LIN {X 0,Y 530.972,Z 518.34,A -85,B 0,C 180,E1 -4177.507,E2 -4177.507} C_VEL
LIN {X 0,Y 530.988,Z 518.342,A -85,B 0,C 180,E1 -4180.433,E2 -4180.433} C_VEL
LIN {X 0,Y 530.965,Z 518.332,A -85,B 0,C 180,E1 -4183.281,E2 -4183.281} C_VEL
LIN {X 0,Y 530.993,Z 518.336,A -85,B 0,C 180,E1 -4185.621,E2 -4185.621} C_VEL
LIN {X 0,Y 531.003,Z 518.341,A -85,B 0,C 180,E1 -4188.565,E2 -4188.565} C_VEL
LIN {X 0,Y 530.963,Z 518.337,A -85,B 0,C 180,E1 -4191.529,E2 -4191.529} C_VEL
LIN {X 0,Y 530.959,Z 518.348,A -85,B 0,C 180,E1 -4194.38,E2 -4194.38} C_VEL
LIN {X 0,Y 530.972,Z 518.342,A -85,B 0,C 180,E1 -4197.133,E2 -4197.133} C_VEL
LIN {X 0,Y 530.975,Z 518.34,A -85,B 0,C 180,E1 -4199.803,E2 -4199.803} C_VEL
LIN {X 0,Y 531.018,Z 518.341,A -85,B 0,C 180,E1 -4202.467,E2 -4202.467} C_VEL
LIN {X 0,Y 531,Z 518.339,A -85,B 0,C 180,E1 -4204.942,E2 -4204.942} C_VEL
LIN {X 0,Y 530.977,Z 518.342,A -85,B 0,C 180,E1 -4208.246,E2 -4208.246} C_VEL
LIN {X 0,Y 531.049,Z 518.493,A -85,B 0,C 180,E1 -4209.545,E2 -4209.545} C_VEL
LIN {X 0,Y 531.712,Z 523.199,A -85,B 0,C 180,E1 -4210.505,E2 -4210.505} C_VEL
LIN {X 0,Y 531.398,Z 538.775,A -85,B 0,C 180,E1 -4213.48,E2 -4213.48} C_VEL
LIN {X 0,Y 531.21,Z 547.447,A -85,B 0,C 180,E1 -4215.07,E2 -4215.07} C_VEL
LIN {X 0,Y 531.552,Z 549.944,A -85,B 0,C 180,E1 -4215.153,E2 -4215.153} C_VEL
LIN {X 0,Y 532.809,Z 556.748,A -85,B 0,C 180,E1 -4215.283,E2 -4215.283} C_VEL
LIN {X 0,Y 532.432,Z 654.187,A -85,B 0,C 180,E1 -4216.619,E2 -4216.619} C_VEL
LIN {X 0,Y 532.263,Z 667.399,A -85,B 0,C 180,E1 -4216.955,E2 -4216.955} C_VEL
LIN {X 0,Y 532.009,Z 679.508,A -85,B 0,C 180,E1 -4217.41,E2 -4217.41} C_VEL
LIN {X 0,Y 531.827,Z 691.228,A -85,B 0,C 180,E1 -4218.006,E2 -4218.006} C_VEL
LIN {X 0,Y 531.578,Z 702.617,A -85,B 0,C 180,E1 -4218.754,E2 -4218.754} C_VEL
LIN {X 0,Y 531.28,Z 713.098,A -85,B 0,C 180,E1 -4219.616,E2 -4219.616} C_VEL
LIN {X 0,Y 531.071,Z 721.693,A -85,B 0,C 180,E1 -4220.478,E2 -4220.478} C_VEL
LIN {X 0,Y 530.892,Z 729.61,A -85,B 0,C 180,E1 -4221.435,E2 -4221.435} C_VEL
LIN {X 0,Y 530.69,Z 737.354,A -85,B 0,C 180,E1 -4222.581,E2 -4222.581} C_VEL
LIN {X 0,Y 530.607,Z 744.463,A -85,B 0,C 180,E1 -4223.917,E2 -4223.917} C_VEL
LIN {X 0,Y 530.459,Z 749.203,A -85,B 0,C 180,E1 -4225.059,E2 -4225.059} C_VEL
LIN {X 0,Y 530.516,Z 752.832,A -85,B 0,C 180,E1 -4226.201,E2 -4226.201} C_VEL
LIN {X 0,Y 530.457,Z 754.71,A -85,B 0,C 180,E1 -4226.961,E2 -4226.961} C_VEL
LIN {X 0,Y 530.411,Z 756.13,A -85,B 0,C 180,E1 -4227.721,E2 -4227.721} C_VEL
LIN {X 0,Y 530.344,Z 757.757,A -85,B 0,C 180,E1 -4229.24,E2 -4229.24} C_VEL
LIN {X 0,Y 530.343,Z 757.996,A -85,B 0,C 180,E1 -4229.999,E2 -4229.999} C_VEL
LIN {X 0,Y 530.344,Z 757.814,A -85,B 0,C 180,E1 -4230.759,E2 -4230.759} C_VEL
LIN {X 0,Y 530.411,Z 756.265,A -85,B 0,C 180,E1 -4232.277,E2 -4232.277} C_VEL
LIN {X 0,Y 530.457,Z 754.903,A -85,B 0,C 180,E1 -4233.037,E2 -4233.037} C_VEL
LIN {X 0,Y 530.523,Z 752.022,A -85,B 0,C 180,E1 -4234.178,E2 -4234.178} C_VEL
LIN {X 0,Y 530.523,Z 748.12,A -85,B 0,C 180,E1 -4235.32,E2 -4235.32} C_VEL
LIN {X 0,Y 530.592,Z 742.537,A -85,B 0,C 180,E1 -4236.575,E2 -4236.575} C_VEL
LIN {X 0,Y 530.757,Z 735.529,A -85,B 0,C 180,E1 -4237.8,E2 -4237.8} C_VEL
LIN {X 0,Y 530.927,Z 727.344,A -85,B 0,C 180,E1 -4238.947,E2 -4238.947} C_VEL
LIN {X 0,Y 531.104,Z 718.973,A -85,B 0,C 180,E1 -4239.905,E2 -4239.905} C_VEL
LIN {X 0,Y 531.417,Z 708.669,A -85,B 0,C 180,E1 -4240.862,E2 -4240.862} C_VEL
LIN {X 0,Y 531.692,Z 698.123,A -85,B 0,C 180,E1 -4241.651,E2 -4241.651} C_VEL
LIN {X 0,Y 531.871,Z 687.286,A -85,B 0,C 180,E1 -4242.302,E2 -4242.302} C_VEL
LIN {X 0,Y 532.145,Z 674.78,A -85,B 0,C 180,E1 -4242.877,E2 -4242.877} C_VEL
LIN {X 0,Y 532.325,Z 661.344,A -85,B 0,C 180,E1 -4243.309,E2 -4243.309} C_VEL
LIN {X 0,Y 532.502,Z 647.993,A -85,B 0,C 180,E1 -4243.572,E2 -4243.572} C_VEL
LIN {X 0,Y 532.735,Z 556.435,A -85,B 0,C 180,E1 -4244.814,E2 -4244.814} C_VEL
LIN {X 0,Y 531.26,Z 547.806,A -85,B 0,C 180,E1 -4244.989,E2 -4244.989} C_VEL
LIN {X 0,Y 531.226,Z 545.512,A -85,B 0,C 180,E1 -4245.342,E2 -4245.342} C_VEL
LIN {X 0,Y 531.548,Z 530.014,A -85,B 0,C 180,E1 -4248.281,E2 -4248.281} C_VEL
LIN {X 0,Y 531.674,Z 522.635,A -85,B 0,C 180,E1 -4249.698,E2 -4249.698} C_VEL
LIN {X 0,Y 531.04,Z 518.404,A -85,B 0,C 180,E1 -4250.58,E2 -4250.58} C_VEL
LIN {X 0,Y 530.998,Z 518.339,A -85,B 0,C 180,E1 -4254.041,E2 -4254.041} C_VEL
LIN {X 0,Y 531.005,Z 518.336,A -85,B 0,C 180,E1 -4256.743,E2 -4256.743} C_VEL
LIN {X 0,Y 530.982,Z 518.342,A -85,B 0,C 180,E1 -4259.322,E2 -4259.322} C_VEL
LIN {X 0,Y 530.979,Z 518.34,A -85,B 0,C 180,E1 -4262.102,E2 -4262.102} C_VEL
LIN {X 0,Y 530.987,Z 518.341,A -85,B 0,C 180,E1 -4264.853,E2 -4264.853} C_VEL
LIN {X 0,Y 530.965,Z 518.349,A -85,B 0,C 180,E1 -4267.507,E2 -4267.507} C_VEL
LIN {X 0,Y 530.982,Z 518.336,A -85,B 0,C 180,E1 -4270.432,E2 -4270.432} C_VEL
LIN {X 0,Y 530.968,Z 518.348,A -85,B 0,C 180,E1 -4273.281,E2 -4273.281} C_VEL
LIN {X 0,Y 530.984,Z 518.344,A -85,B 0,C 180,E1 -4275.62,E2 -4275.62} C_VEL
LIN {X 0,Y 531.003,Z 518.336,A -85,B 0,C 180,E1 -4278.565,E2 -4278.565} C_VEL
LIN {X 0,Y 530.964,Z 518.342,A -85,B 0,C 180,E1 -4281.345,E2 -4281.345} C_VEL
LIN {X 0,Y 530.978,Z 518.339,A -85,B 0,C 180,E1 -4284.382,E2 -4284.382} C_VEL
LIN {X 0,Y 530.97,Z 518.344,A -85,B 0,C 180,E1 -4287.133,E2 -4287.133} C_VEL
LIN {X 0,Y 530.981,Z 518.343,A -85,B 0,C 180,E1 -4289.804,E2 -4289.804} C_VEL
LIN {X 0,Y 531.012,Z 518.332,A -85,B 0,C 180,E1 -4292.466,E2 -4292.466} C_VEL
LIN {X 0,Y 531.002,Z 518.338,A -85,B 0,C 180,E1 -4294.942,E2 -4294.942} C_VEL
LIN {X 0,Y 530.965,Z 518.339,A -85,B 0,C 180,E1 -4298.246,E2 -4298.246} C_VEL
LIN {X 0,Y 530.991,Z 518.337,A -85,B 0,C 180,E1 -4300.677,E2 -4300.677} C_VEL
LIN {X 0,Y 530.987,Z 518.339,A -85,B 0,C 180,E1 -4303.071,E2 -4303.071} C_VEL
LIN {X 0,Y 531.012,Z 518.34,A -85,B 0,C 180,E1 -4305.436,E2 -4305.436} C_VEL
LIN {X 0,Y 531.029,Z 518.331,A -85,B 0,C 180,E1 -4308.549,E2 -4308.549} C_VEL
LIN {X 0,Y 531.053,Z 518.337,A -85,B 0,C 180,E1 -4311.629,E2 -4311.629} C_VEL
LIN {X 0,Y 531.117,Z 518.321,A -85,B 0,C 180,E1 -4314.685,E2 -4314.685} C_VEL
LIN {X 0,Y 531.133,Z 518.325,A -85,B 0,C 180,E1 -4317.725,E2 -4317.725} C_VEL
LIN {X 0,Y 531.148,Z 518.318,A -85,B 0,C 180,E1 -4320.758,E2 -4320.758} C_VEL
LIN {X 0,Y 531.102,Z 518.323,A -85,B 0,C 180,E1 -4323.034,E2 -4323.034} C_VEL
LIN {X 0,Y 531.077,Z 518.329,A -85,B 0,C 180,E1 -4326.077,E2 -4326.077} C_VEL
LIN {X 0,Y 531.025,Z 518.335,A -85,B 0,C 180,E1 -4329.138,E2 -4329.138} C_VEL
LIN {X 0,Y 531.033,Z 518.333,A -85,B 0,C 180,E1 -4332.225,E2 -4332.225} C_VEL
LIN {X 0,Y 530.989,Z 518.342,A -85,B 0,C 180,E1 -4335.35,E2 -4335.35} C_VEL
LIN {X 0,Y 531.009,Z 518.343,A -85,B 0,C 180,E1 -4337.723,E2 -4337.723} C_VEL
LIN {X 0,Y 530.995,Z 518.337,A -85,B 0,C 180,E1 -4340.938,E2 -4340.938} C_VEL
LIN {X 0,Y 530.973,Z 518.341,A -85,B 0,C 180,E1 -4344.225,E2 -4344.225} C_VEL
LIN {X 0,Y 531.005,Z 518.333,A -85,B 0,C 180,E1 -4346.744,E2 -4346.744} C_VEL
LIN {X 0,Y 530.976,Z 518.344,A -85,B 0,C 180,E1 -4349.323,E2 -4349.323} C_VEL
LIN {X 0,Y 530.975,Z 518.342,A -85,B 0,C 180,E1 -4352.104,E2 -4352.104} C_VEL
LIN {X 0,Y 530.986,Z 518.337,A -85,B 0,C 180,E1 -4354.855,E2 -4354.855} C_VEL
LIN {X 0,Y 530.961,Z 518.342,A -85,B 0,C 180,E1 -4357.508,E2 -4357.508} C_VEL
LIN {X 0,Y 530.98,Z 518.339,A -85,B 0,C 180,E1 -4360.433,E2 -4360.433} C_VEL
LIN {X 0,Y 530.959,Z 518.341,A -85,B 0,C 180,E1 -4363.282,E2 -4363.282} C_VEL
LIN {X 0,Y 530.984,Z 518.347,A -85,B 0,C 180,E1 -4365.622,E2 -4365.622} C_VEL
LIN {X 0,Y 531.004,Z 518.336,A -85,B 0,C 180,E1 -4368.567,E2 -4368.567} C_VEL
LIN {X 0,Y 530.966,Z 518.342,A -85,B 0,C 180,E1 -4371.347,E2 -4371.347} C_VEL
LIN {X 0,Y 530.974,Z 518.341,A -85,B 0,C 180,E1 -4374.383,E2 -4374.383} C_VEL
LIN {X 0,Y 530.971,Z 518.338,A -85,B 0,C 180,E1 -4377.135,E2 -4377.135} C_VEL
LIN {X 0,Y 530.968,Z 518.329,A -85,B 0,C 180,E1 -4379.804,E2 -4379.804} C_VEL
LIN {X 0,Y 531.016,Z 518.334,A -85,B 0,C 180,E1 -4382.468,E2 -4382.468} C_VEL
LIN {X 0,Y 531.006,Z 518.336,A -85,B 0,C 180,E1 -4384.943,E2 -4384.943} C_VEL
LIN {X 0,Y 531.017,Z 518.525,A -85,B 0,C 180,E1 -4385.967,E2 -4385.967} C_VEL
LIN {X 0,Y 532.382,Z 526.216,A -85,B 0,C 180,E1 -4387.287,E2 -4387.287} C_VEL
LIN {X 0,Y 531.99,Z 544.026,A -85,B 0,C 180,E1 -4390.113,E2 -4390.113} C_VEL
LIN {X 0,Y 531.618,Z 561.828,A -85,B 0,C 180,E1 -4392.895,E2 -4392.895} C_VEL
LIN {X 0,Y 531.386,Z 575.727,A -85,B 0,C 180,E1 -4395.018,E2 -4395.018} C_VEL
LIN {X 0,Y 531.936,Z 579.534,A -85,B 0,C 180,E1 -4395.119,E2 -4395.119} C_VEL
LIN {X 0,Y 532.852,Z 586.52,A -85,B 0,C 180,E1 -4395.24,E2 -4395.24} C_VEL
LIN {X 0,Y 532.447,Z 683.947,A -85,B 0,C 180,E1 -4396.573,E2 -4396.573} C_VEL
LIN {X 0,Y 532.241,Z 697.212,A -85,B 0,C 180,E1 -4396.907,E2 -4396.907} C_VEL
LIN {X 0,Y 532.003,Z 710.499,A -85,B 0,C 180,E1 -4397.411,E2 -4397.411} C_VEL
LIN {X 0,Y 531.803,Z 721.954,A -85,B 0,C 180,E1 -4398.007,E2 -4398.007} C_VEL
LIN {X 0,Y 531.557,Z 733.204,A -85,B 0,C 180,E1 -4398.755,E2 -4398.755} C_VEL
LIN {X 0,Y 531.267,Z 743.612,A -85,B 0,C 180,E1 -4399.617,E2 -4399.617} C_VEL
LIN {X 0,Y 531.06,Z 752.121,A -85,B 0,C 180,E1 -4400.479,E2 -4400.479} C_VEL
LIN {X 0,Y 530.886,Z 759.966,A -85,B 0,C 180,E1 -4401.436,E2 -4401.436} C_VEL
LIN {X 0,Y 530.684,Z 767.626,A -85,B 0,C 180,E1 -4402.582,E2 -4402.582} C_VEL
LIN {X 0,Y 530.602,Z 774.682,A -85,B 0,C 180,E1 -4403.918,E2 -4403.918} C_VEL
LIN {X 0,Y 530.459,Z 779.375,A -85,B 0,C 180,E1 -4405.06,E2 -4405.06} C_VEL
LIN {X 0,Y 530.516,Z 782.962,A -85,B 0,C 180,E1 -4406.203,E2 -4406.203} C_VEL
LIN {X 0,Y 530.457,Z 784.811,A -85,B 0,C 180,E1 -4406.963,E2 -4406.963} C_VEL
LIN {X 0,Y 530.41,Z 786.197,A -85,B 0,C 180,E1 -4407.723,E2 -4407.723} C_VEL
LIN {X 0,Y 530.344,Z 787.786,A -85,B 0,C 180,E1 -4409.241,E2 -4409.241} C_VEL
LIN {X 0,Y 530.342,Z 788,A -85,B 0,C 180,E1 -4410.001,E2 -4410.001} C_VEL
LIN {X 0,Y 530.361,Z 787.181,A -85,B 0,C 180,E1 -4411.519,E2 -4411.519} C_VEL
LIN {X 0,Y 530.41,Z 786.193,A -85,B 0,C 180,E1 -4412.279,E2 -4412.279} C_VEL
LIN {X 0,Y 530.457,Z 784.805,A -85,B 0,C 180,E1 -4413.039,E2 -4413.039} C_VEL
LIN {X 0,Y 530.522,Z 781.892,A -85,B 0,C 180,E1 -4414.179,E2 -4414.179} C_VEL
LIN {X 0,Y 530.525,Z 777.947,A -85,B 0,C 180,E1 -4415.321,E2 -4415.321} C_VEL
LIN {X 0,Y 530.599,Z 772.261,A -85,B 0,C 180,E1 -4416.582,E2 -4416.582} C_VEL
LIN {X 0,Y 530.759,Z 765.231,A -85,B 0,C 180,E1 -4417.801,E2 -4417.801} C_VEL
LIN {X 0,Y 530.931,Z 756.987,A -85,B 0,C 180,E1 -4418.949,E2 -4418.949} C_VEL
LIN {X 0,Y 531.14,Z 748.533,A -85,B 0,C 180,E1 -4419.906,E2 -4419.906} C_VEL
LIN {X 0,Y 531.413,Z 738.084,A -85,B 0,C 180,E1 -4420.863,E2 -4420.863} C_VEL
LIN {X 0,Y 531.694,Z 727.344,A -85,B 0,C 180,E1 -4421.656,E2 -4421.656} C_VEL
LIN {X 0,Y 531.906,Z 716.395,A -85,B 0,C 180,E1 -4422.302,E2 -4422.302} C_VEL
LIN {X 0,Y 532.133,Z 704.752,A -85,B 0,C 180,E1 -4422.83,E2 -4422.83} C_VEL
LIN {X 0,Y 532.333,Z 691.301,A -85,B 0,C 180,E1 -4423.262,E2 -4423.262} C_VEL
LIN {X 0,Y 532.485,Z 678.003,A -85,B 0,C 180,E1 -4423.525,E2 -4423.525} C_VEL
LIN {X 0,Y 532.711,Z 584.395,A -85,B 0,C 180,E1 -4424.793,E2 -4424.793} C_VEL
LIN {X 0,Y 531.369,Z 576.167,A -85,B 0,C 180,E1 -4424.954,E2 -4424.954} C_VEL
LIN {X 0,Y 531.33,Z 575.003,A -85,B 0,C 180,E1 -4425.075,E2 -4425.075} C_VEL
LIN {X 0,Y 531.8,Z 554.095,A -85,B 0,C 180,E1 -4428.308,E2 -4428.308} C_VEL
LIN {X 0,Y 532.199,Z 533.839,A -85,B 0,C 180,E1 -4431.498,E2 -4431.498} C_VEL
LIN {X 0,Y 532.425,Z 526.21,A -85,B 0,C 180,E1 -4432.713,E2 -4432.713} C_VEL
LIN {X 0,Y 531.005,Z 518.517,A -85,B 0,C 180,E1 -4434.043,E2 -4434.043} C_VEL
LIN {X 0,Y 531.008,Z 518.34,A -85,B 0,C 180,E1 -4436.744,E2 -4436.744} C_VEL
LIN {X 0,Y 530.985,Z 518.328,A -85,B 0,C 180,E1 -4439.323,E2 -4439.323} C_VEL
LIN {X 0,Y 530.97,Z 518.348,A -85,B 0,C 180,E1 -4442.101,E2 -4442.101} C_VEL
LIN {X 0,Y 530.974,Z 518.341,A -85,B 0,C 180,E1 -4444.851,E2 -4444.851} C_VEL
LIN {X 0,Y 530.97,Z 518.342,A -85,B 0,C 180,E1 -4447.508,E2 -4447.508} C_VEL
LIN {X 0,Y 530.986,Z 518.342,A -85,B 0,C 180,E1 -4450.433,E2 -4450.433} C_VEL
LIN {X 0,Y 530.97,Z 518.342,A -85,B 0,C 180,E1 -4453.282,E2 -4453.282} C_VEL
LIN {X 0,Y 530.993,Z 518.343,A -85,B 0,C 180,E1 -4455.621,E2 -4455.621} C_VEL
LIN {X 0,Y 531.005,Z 518.338,A -85,B 0,C 180,E1 -4458.565,E2 -4458.565} C_VEL
LIN {X 0,Y 530.963,Z 518.345,A -85,B 0,C 180,E1 -4461.53,E2 -4461.53} C_VEL
LIN {X 0,Y 530.986,Z 518.341,A -85,B 0,C 180,E1 -4464.382,E2 -4464.382} C_VEL
LIN {X 0,Y 530.975,Z 518.342,A -85,B 0,C 180,E1 -4467.134,E2 -4467.134} C_VEL
LIN {X 0,Y 530.974,Z 518.349,A -85,B 0,C 180,E1 -4469.803,E2 -4469.803} C_VEL
LIN {X 0,Y 531.016,Z 518.34,A -85,B 0,C 180,E1 -4472.468,E2 -4472.468} C_VEL
LIN {X 0,Y 531.083,Z 518.57,A -85,B 0,C 180,E1 -4474.181,E2 -4474.181} C_VEL
LIN {X 0,Y 532.508,Z 527.2,A -85,B 0,C 180,E1 -4475.353,E2 -4475.353} C_VEL
LIN {X 0,Y 532.305,Z 548.46,A -85,B 0,C 180,E1 -4478.101,E2 -4478.101} C_VEL
LIN {X 0,Y 531.95,Z 571.078,A -85,B 0,C 180,E1 -4481.114,E2 -4481.114} C_VEL
LIN {X 0,Y 531.744,Z 586.094,A -85,B 0,C 180,E1 -4483.096,E2 -4483.096} C_VEL
LIN {X 0,Y 531.35,Z 607.645,A -85,B 0,C 180,E1 -4486.032,E2 -4486.032} C_VEL
LIN {X 0,Y 531.097,Z 631.056,A -85,B 0,C 180,E1 -4489.179,E2 -4489.179} C_VEL
LIN {X 0,Y 531.686,Z 639.829,A -85,B 0,C 180,E1 -4489.336,E2 -4489.336} C_VEL
LIN {X 0,Y 531.503,Z 702.519,A -85,B 0,C 180,E1 -4490.198,E2 -4490.198} C_VEL
LIN {X 0,Y 531.443,Z 713.787,A -85,B 0,C 180,E1 -4490.509,E2 -4490.509} C_VEL
LIN {X 0,Y 531.308,Z 724.494,A -85,B 0,C 180,E1 -4490.963,E2 -4490.963} C_VEL
LIN {X 0,Y 531.121,Z 734.267,A -85,B 0,C 180,E1 -4491.535,E2 -4491.535} C_VEL
LIN {X 0,Y 530.915,Z 744.061,A -85,B 0,C 180,E1 -4492.297,E2 -4492.297} C_VEL
LIN {X 0,Y 530.769,Z 752.567,A -85,B 0,C 180,E1 -4493.156,E2 -4493.156} C_VEL
LIN {X 0,Y 530.723,Z 759.945,A -85,B 0,C 180,E1 -4494.109,E2 -4494.109} C_VEL
LIN {X 0,Y 530.564,Z 765.69,A -85,B 0,C 180,E1 -4495.061,E2 -4495.061} C_VEL
LIN {X 0,Y 530.539,Z 770.879,A -85,B 0,C 180,E1 -4496.202,E2 -4496.202} C_VEL
LIN {X 0,Y 530.506,Z 773.479,A -85,B 0,C 180,E1 -4496.962,E2 -4496.962} C_VEL
LIN {X 0,Y 530.413,Z 775.428,A -85,B 0,C 180,E1 -4497.722,E2 -4497.722} C_VEL
LIN {X 0,Y 530.358,Z 776.826,A -85,B 0,C 180,E1 -4498.481,E2 -4498.481} C_VEL
LIN {X 0,Y 530.339,Z 777.679,A -85,B 0,C 180,E1 -4499.241,E2 -4499.241} C_VEL
LIN {X 0,Y 530.341,Z 777.997,A -85,B 0,C 180,E1 -4500,E2 -4500} C_VEL
LIN {X 0,Y 530.342,Z 777.758,A -85,B 0,C 180,E1 -4500.759,E2 -4500.759} C_VEL
LIN {X 0,Y 530.36,Z 776.962,A -85,B 0,C 180,E1 -4501.519,E2 -4501.519} C_VEL
LIN {X 0,Y 530.41,Z 775.62,A -85,B 0,C 180,E1 -4502.278,E2 -4502.278} C_VEL
LIN {X 0,Y 530.497,Z 772.547,A -85,B 0,C 180,E1 -4503.418,E2 -4503.418} C_VEL
LIN {X 0,Y 530.537,Z 768.012,A -85,B 0,C 180,E1 -4504.559,E2 -4504.559} C_VEL
LIN {X 0,Y 530.6,Z 762.96,A -85,B 0,C 180,E1 -4505.511,E2 -4505.511} C_VEL
LIN {X 0,Y 530.759,Z 756.287,A -85,B 0,C 180,E1 -4506.483,E2 -4506.483} C_VEL
LIN {X 0,Y 530.853,Z 748.049,A -85,B 0,C 180,E1 -4507.417,E2 -4507.417} C_VEL
LIN {X 0,Y 531.02,Z 739.419,A -85,B 0,C 180,E1 -4508.18,E2 -4508.18} C_VEL
LIN {X 0,Y 531.205,Z 729.638,A -85,B 0,C 180,E1 -4508.847,E2 -4508.847} C_VEL
LIN {X 0,Y 531.352,Z 719.194,A -85,B 0,C 180,E1 -4509.373,E2 -4509.373} C_VEL
LIN {X 0,Y 531.471,Z 708.225,A -85,B 0,C 180,E1 -4509.755,E2 -4509.755} C_VEL
LIN {X 0,Y 531.57,Z 696.598,A -85,B 0,C 180,E1 -4509.993,E2 -4509.993} C_VEL
LIN {X 0,Y 531.622,Z 636.669,A -85,B 0,C 180,E1 -4510.798,E2 -4510.798} C_VEL
LIN {X 0,Y 531.092,Z 631.352,A -85,B 0,C 180,E1 -4510.894,E2 -4510.894} C_VEL
LIN {X 0,Y 531.082,Z 629.77,A -85,B 0,C 180,E1 -4511.063,E2 -4511.063} C_VEL
LIN {X 0,Y 531.415,Z 605.491,A -85,B 0,C 180,E1 -4514.358,E2 -4514.358} C_VEL
LIN {X 0,Y 531.833,Z 582.549,A -85,B 0,C 180,E1 -4517.496,E2 -4517.496} C_VEL
LIN {X 0,Y 532.23,Z 559.842,A -85,B 0,C 180,E1 -4520.556,E2 -4520.556} C_VEL
LIN {X 0,Y 532.64,Z 538.189,A -85,B 0,C 180,E1 -4523.524,E2 -4523.524} C_VEL
LIN {X 0,Y 532.753,Z 527.599,A -85,B 0,C 180,E1 -4524.97,E2 -4524.97} C_VEL
LIN {X 0,Y 531.041,Z 518.503,A -85,B 0,C 180,E1 -4526.318,E2 -4526.318} C_VEL
LIN {X 0,Y 530.993,Z 518.341,A -85,B 0,C 180,E1 -4529.126,E2 -4529.126} C_VEL
LIN {X 0,Y 530.972,Z 518.342,A -85,B 0,C 180,E1 -4529.531,E2 -4529.531} C_VEL
LIN {X 0,Y 530.289,Z 518.433,A -85,B 0,C 180,E1 -4530.164,E2 -4530.164} C_VEL
LIN {X 0,Y 527.431,Z 518.789,A -85,B 0,C 180,E1 -4531.192,E2 -4531.192} C_VEL
LIN {X 0,Y 525.029,Z 519.088,A -85,B 0,C 180,E1 -4532.02,E2 -4532.02} C_VEL
LIN {X 0,Y 524.005,Z 519.214,A -85,B 0,C 180,E1 -4532.659,E2 -4532.659} C_VEL
LIN {X 0,Y 523.925,Z 519.221,A -85,B 0,C 180,E1 -4532.875,E2 -4532.875} C_VEL
LIN {X 0,Y 523.941,Z 519.217,A -85,B 0,C 180,E1 -4535.225,E2 -4535.225} C_VEL
LIN {X 0,Y 523.922,Z 519.222,A -85,B 0,C 180,E1 -4538.102,E2 -4538.102} C_VEL
LIN {X 0,Y 523.946,Z 519.209,A -85,B 0,C 180,E1 -4541.092,E2 -4541.092} C_VEL
LIN {X 0,Y 523.942,Z 519.211,A -85,B 0,C 180,E1 -4544.228,E2 -4544.228} C_VEL
LIN {X 0,Y 523.93,Z 519.222,A -85,B 0,C 180,E1 -4546.834,E2 -4546.834} C_VEL
LIN {X 0,Y 523.947,Z 519.214,A -85,B 0,C 180,E1 -4548.908,E2 -4548.908} C_VEL
LIN {X 0,Y 523.921,Z 519.216,A -85,B 0,C 180,E1 -4551.898,E2 -4551.898} C_VEL
LIN {X 0,Y 523.929,Z 519.219,A -85,B 0,C 180,E1 -4554.911,E2 -4554.911} C_VEL
LIN {X 0,Y 523.94,Z 519.216,A -85,B 0,C 180,E1 -4557.679,E2 -4557.679} C_VEL
LIN {X 0,Y 523.959,Z 519.221,A -85,B 0,C 180,E1 -4560.676,E2 -4560.676} C_VEL
LIN {X 0,Y 523.979,Z 519.212,A -85,B 0,C 180,E1 -4563.728,E2 -4563.728} C_VEL
LIN {X 0,Y 523.932,Z 519.217,A -85,B 0,C 180,E1 -4566.27,E2 -4566.27} C_VEL
LIN {X 0,Y 523.992,Z 519.334,A -85,B 0,C 180,E1 -4569.385,E2 -4569.385} C_VEL
LIN {X 0,Y 524.769,Z 524.408,A -85,B 0,C 180,E1 -4570.438,E2 -4570.438} C_VEL
LIN {X 0,Y 524.356,Z 541.046,A -85,B 0,C 180,E1 -4573.652,E2 -4573.652} C_VEL
LIN {X 0,Y 524.229,Z 547.516,A -85,B 0,C 180,E1 -4574.854,E2 -4574.854} C_VEL
LIN {X 0,Y 524.589,Z 550.039,A -85,B 0,C 180,E1 -4574.949,E2 -4574.949} C_VEL
LIN {X 0,Y 525.958,Z 557.678,A -85,B 0,C 180,E1 -4575.096,E2 -4575.096} C_VEL
LIN {X 0,Y 525.546,Z 654.42,A -85,B 0,C 180,E1 -4576.441,E2 -4576.441} C_VEL
LIN {X 0,Y 525.372,Z 667.621,A -85,B 0,C 180,E1 -4576.781,E2 -4576.781} C_VEL
LIN {X 0,Y 525.105,Z 679.723,A -85,B 0,C 180,E1 -4577.241,E2 -4577.241} C_VEL
LIN {X 0,Y 524.901,Z 690.663,A -85,B 0,C 180,E1 -4577.8,E2 -4577.8} C_VEL
LIN {X 0,Y 524.634,Z 701.514,A -85,B 0,C 180,E1 -4578.505,E2 -4578.505} C_VEL
LIN {X 0,Y 524.319,Z 712.216,A -85,B 0,C 180,E1 -4579.379,E2 -4579.379} C_VEL
LIN {X 0,Y 524.061,Z 721.842,A -85,B 0,C 180,E1 -4580.349,E2 -4580.349} C_VEL
LIN {X 0,Y 523.86,Z 729.724,A -85,B 0,C 180,E1 -4581.319,E2 -4581.319} C_VEL
LIN {X 0,Y 523.637,Z 737.43,A -85,B 0,C 180,E1 -4582.48,E2 -4582.48} C_VEL
LIN {X 0,Y 523.519,Z 744.5,A -85,B 0,C 180,E1 -4583.834,E2 -4583.834} C_VEL
LIN {X 0,Y 523.384,Z 749.231,A -85,B 0,C 180,E1 -4584.992,E2 -4584.992} C_VEL
LIN {X 0,Y 523.444,Z 752.839,A -85,B 0,C 180,E1 -4586.15,E2 -4586.15} C_VEL
LIN {X 0,Y 523.368,Z 754.712,A -85,B 0,C 180,E1 -4586.92,E2 -4586.92} C_VEL
LIN {X 0,Y 523.335,Z 756.13,A -85,B 0,C 180,E1 -4587.69,E2 -4587.69} C_VEL
LIN {X 0,Y 523.25,Z 757.757,A -85,B 0,C 180,E1 -4589.23,E2 -4589.23} C_VEL
LIN {X 0,Y 523.247,Z 757.997,A -85,B 0,C 180,E1 -4589.999,E2 -4589.999} C_VEL
LIN {X 0,Y 523.25,Z 757.814,A -85,B 0,C 180,E1 -4590.769,E2 -4590.769} C_VEL
LIN {X 0,Y 523.335,Z 756.263,A -85,B 0,C 180,E1 -4592.308,E2 -4592.308} C_VEL
LIN {X 0,Y 523.368,Z 754.901,A -85,B 0,C 180,E1 -4593.078,E2 -4593.078} C_VEL
LIN {X 0,Y 523.441,Z 752.025,A -85,B 0,C 180,E1 -4594.234,E2 -4594.234} C_VEL
LIN {X 0,Y 523.462,Z 748.133,A -85,B 0,C 180,E1 -4595.392,E2 -4595.392} C_VEL
LIN {X 0,Y 523.516,Z 743.024,A -85,B 0,C 180,E1 -4596.573,E2 -4596.573} C_VEL
LIN {X 0,Y 523.664,Z 736.83,A -85,B 0,C 180,E1 -4597.712,E2 -4597.712} C_VEL
LIN {X 0,Y 523.876,Z 728.94,A -85,B 0,C 180,E1 -4598.874,E2 -4598.874} C_VEL
LIN {X 0,Y 524.097,Z 719.123,A -85,B 0,C 180,E1 -4600.039,E2 -4600.039} C_VEL
LIN {X 0,Y 524.444,Z 708.833,A -85,B 0,C 180,E1 -4601.008,E2 -4601.008} C_VEL
LIN {X 0,Y 524.725,Z 698.74,A -85,B 0,C 180,E1 -4601.778,E2 -4601.778} C_VEL
LIN {X 0,Y 524.942,Z 687.481,A -85,B 0,C 180,E1 -4602.467,E2 -4602.467} C_VEL
LIN {X 0,Y 525.249,Z 674.96,A -85,B 0,C 180,E1 -4603.049,E2 -4603.049} C_VEL
LIN {X 0,Y 525.422,Z 661.522,A -85,B 0,C 180,E1 -4603.487,E2 -4603.487} C_VEL
LIN {X 0,Y 525.618,Z 648.153,A -85,B 0,C 180,E1 -4603.753,E2 -4603.753} C_VEL
LIN {X 0,Y 525.846,Z 557.035,A -85,B 0,C 180,E1 -4605.006,E2 -4605.006} C_VEL
LIN {X 0,Y 524.28,Z 547.869,A -85,B 0,C 180,E1 -4605.205,E2 -4605.205} C_VEL
LIN {X 0,Y 524.223,Z 545.692,A -85,B 0,C 180,E1 -4605.552,E2 -4605.552} C_VEL
LIN {X 0,Y 524.583,Z 531.329,A -85,B 0,C 180,E1 -4608.31,E2 -4608.31} C_VEL
LIN {X 0,Y 524.636,Z 523.164,A -85,B 0,C 180,E1 -4609.902,E2 -4609.902} C_VEL
LIN {X 0,Y 523.979,Z 519.256,A -85,B 0,C 180,E1 -4610.742,E2 -4610.742} C_VEL
LIN {X 0,Y 523.963,Z 519.215,A -85,B 0,C 180,E1 -4614.203,E2 -4614.203} C_VEL
LIN {X 0,Y 523.953,Z 519.218,A -85,B 0,C 180,E1 -4617.132,E2 -4617.132} C_VEL
LIN {X 0,Y 523.942,Z 519.218,A -85,B 0,C 180,E1 -4619.755,E2 -4619.755} C_VEL
LIN {X 0,Y 523.939,Z 519.216,A -85,B 0,C 180,E1 -4622.448,E2 -4622.448} C_VEL
LIN {X 0,Y 523.934,Z 519.224,A -85,B 0,C 180,E1 -4625.224,E2 -4625.224} C_VEL
LIN {X 0,Y 523.915,Z 519.22,A -85,B 0,C 180,E1 -4628.101,E2 -4628.101} C_VEL
LIN {X 0,Y 523.959,Z 519.219,A -85,B 0,C 180,E1 -4631.31,E2 -4631.31} C_VEL
LIN {X 0,Y 523.952,Z 519.211,A -85,B 0,C 180,E1 -4634.691,E2 -4634.691} C_VEL
LIN {X 0,Y 523.952,Z 519.217,A -85,B 0,C 180,E1 -4637.881,E2 -4637.881} C_VEL
LIN {X 0,Y 523.955,Z 519.212,A -85,B 0,C 180,E1 -4640.918,E2 -4640.918} C_VEL
LIN {X 0,Y 523.925,Z 519.221,A -85,B 0,C 180,E1 -4643.827,E2 -4643.827} C_VEL
LIN {X 0,Y 523.939,Z 519.216,A -85,B 0,C 180,E1 -4646.635,E2 -4646.635} C_VEL
LIN {X 0,Y 523.958,Z 519.22,A -85,B 0,C 180,E1 -4649.356,E2 -4649.356} C_VEL
LIN {X 0,Y 523.974,Z 519.209,A -85,B 0,C 180,E1 -4652.28,E2 -4652.28} C_VEL
LIN {X 0,Y 523.949,Z 519.214,A -85,B 0,C 180,E1 -4654.581,E2 -4654.581} C_VEL
LIN {X 0,Y 523.91,Z 519.222,A -85,B 0,C 180,E1 -4657.106,E2 -4657.106} C_VEL
LIN {X 0,Y 523.972,Z 519.215,A -85,B 0,C 180,E1 -4659.865,E2 -4659.865} C_VEL
LIN {X 0,Y 523.964,Z 519.212,A -85,B 0,C 180,E1 -4662.837,E2 -4662.837} C_VEL
LIN {X 0,Y 523.969,Z 519.214,A -85,B 0,C 180,E1 -4665.235,E2 -4665.235} C_VEL
LIN {X 0,Y 524.004,Z 519.206,A -85,B 0,C 180,E1 -4668.394,E2 -4668.394} C_VEL
LIN {X 0,Y 524,Z 519.214,A -85,B 0,C 180,E1 -4671.516,E2 -4671.516} C_VEL
LIN {X 0,Y 524.078,Z 519.198,A -85,B 0,C 180,E1 -4674.614,E2 -4674.614} C_VEL
LIN {X 0,Y 524.105,Z 519.201,A -85,B 0,C 180,E1 -4677.694,E2 -4677.694} C_VEL
LIN {X 0,Y 524.118,Z 519.194,A -85,B 0,C 180,E1 -4680.768,E2 -4680.768} C_VEL
LIN {X 0,Y 524.069,Z 519.2,A -85,B 0,C 180,E1 -4683.075,E2 -4683.075} C_VEL
LIN {X 0,Y 524.039,Z 519.205,A -85,B 0,C 180,E1 -4686.159,E2 -4686.159} C_VEL
LIN {X 0,Y 523.993,Z 519.212,A -85,B 0,C 180,E1 -4689.262,E2 -4689.262} C_VEL
LIN {X 0,Y 524.017,Z 519.213,A -85,B 0,C 180,E1 -4691.751,E2 -4691.751} C_VEL
LIN {X 0,Y 523.985,Z 519.211,A -85,B 0,C 180,E1 -4695.053,E2 -4695.053} C_VEL
LIN {X 0,Y 523.957,Z 519.217,A -85,B 0,C 180,E1 -4697.969,E2 -4697.969} C_VEL
LIN {X 0,Y 523.965,Z 519.212,A -85,B 0,C 180,E1 -4700.41,E2 -4700.41} C_VEL
LIN {X 0,Y 523.91,Z 519.219,A -85,B 0,C 180,E1 -4702.894,E2 -4702.894} C_VEL
LIN {X 0,Y 523.949,Z 519.221,A -85,B 0,C 180,E1 -4705.419,E2 -4705.419} C_VEL
LIN {X 0,Y 523.964,Z 519.217,A -85,B 0,C 180,E1 -4707.999,E2 -4707.999} C_VEL
LIN {X 0,Y 523.941,Z 519.215,A -85,B 0,C 180,E1 -4710.856,E2 -4710.856} C_VEL
LIN {X 0,Y 523.957,Z 519.22,A -85,B 0,C 180,E1 -4713.736,E2 -4713.736} C_VEL
LIN {X 0,Y 523.917,Z 519.212,A -85,B 0,C 180,E1 -4716.405,E2 -4716.405} C_VEL
LIN {X 0,Y 523.918,Z 519.22,A -85,B 0,C 180,E1 -4719.085,E2 -4719.085} C_VEL
LIN {X 0,Y 523.952,Z 519.213,A -85,B 0,C 180,E1 -4722.119,E2 -4722.119} C_VEL
LIN {X 0,Y 523.952,Z 519.218,A -85,B 0,C 180,E1 -4725.309,E2 -4725.309} C_VEL
LIN {X 0,Y 523.969,Z 519.213,A -85,B 0,C 180,E1 -4728.688,E2 -4728.688} C_VEL
LIN {X 0,Y 523.922,Z 519.217,A -85,B 0,C 180,E1 -4731.08,E2 -4731.08} C_VEL
LIN {X 0,Y 523.922,Z 519.225,A -85,B 0,C 180,E1 -4733.828,E2 -4733.828} C_VEL
LIN {X 0,Y 523.941,Z 519.212,A -85,B 0,C 180,E1 -4736.637,E2 -4736.637} C_VEL
LIN {X 0,Y 523.955,Z 519.193,A -85,B 0,C 180,E1 -4739.357,E2 -4739.357} C_VEL
LIN {X 0,Y 523.979,Z 519.212,A -85,B 0,C 180,E1 -4742.282,E2 -4742.282} C_VEL
LIN {X 0,Y 523.952,Z 519.208,A -85,B 0,C 180,E1 -4744.582,E2 -4744.582} C_VEL
LIN {X 0,Y 523.986,Z 519.388,A -85,B 0,C 180,E1 -4745.791,E2 -4745.791} C_VEL
LIN {X 0,Y 525.428,Z 527.311,A -85,B 0,C 180,E1 -4747.177,E2 -4747.177} C_VEL
LIN {X 0,Y 525.026,Z 545.12,A -85,B 0,C 180,E1 -4750.042,E2 -4750.042} C_VEL
LIN {X 0,Y 524.582,Z 562.914,A -85,B 0,C 180,E1 -4752.859,E2 -4752.859} C_VEL
LIN {X 0,Y 524.338,Z 575.501,A -85,B 0,C 180,E1 -4754.81,E2 -4754.81} C_VEL
LIN {X 0,Y 524.815,Z 578.845,A -85,B 0,C 180,E1 -4754.905,E2 -4754.905} C_VEL
LIN {X 0,Y 525.976,Z 586.871,A -85,B 0,C 180,E1 -4755.05,E2 -4755.05} C_VEL
LIN {X 0,Y 525.569,Z 683.743,A -85,B 0,C 180,E1 -4756.393,E2 -4756.393} C_VEL
LIN {X 0,Y 525.313,Z 697.007,A -85,B 0,C 180,E1 -4756.732,E2 -4756.732} C_VEL
LIN {X 0,Y 525.054,Z 710.299,A -85,B 0,C 180,E1 -4757.241,E2 -4757.241} C_VEL
LIN {X 0,Y 524.815,Z 722.77,A -85,B 0,C 180,E1 -4757.906,E2 -4757.906} C_VEL
LIN {X 0,Y 524.537,Z 734.362,A -85,B 0,C 180,E1 -4758.7,E2 -4758.7} C_VEL
LIN {X 0,Y 524.244,Z 744.556,A -85,B 0,C 180,E1 -4759.574,E2 -4759.574} C_VEL
LIN {X 0,Y 523.975,Z 753.733,A -85,B 0,C 180,E1 -4760.544,E2 -4760.544} C_VEL
LIN {X 0,Y 523.759,Z 762.675,A -85,B 0,C 180,E1 -4761.707,E2 -4761.707} C_VEL
LIN {X 0,Y 523.583,Z 769.853,A -85,B 0,C 180,E1 -4762.868,E2 -4762.868} C_VEL
LIN {X 0,Y 523.543,Z 776.368,A -85,B 0,C 180,E1 -4764.222,E2 -4764.222} C_VEL
LIN {X 0,Y 523.361,Z 780.679,A -85,B 0,C 180,E1 -4765.379,E2 -4765.379} C_VEL
LIN {X 0,Y 523.443,Z 782.962,A -85,B 0,C 180,E1 -4766.151,E2 -4766.151} C_VEL
LIN {X 0,Y 523.367,Z 784.811,A -85,B 0,C 180,E1 -4766.922,E2 -4766.922} C_VEL
LIN {X 0,Y 523.334,Z 786.197,A -85,B 0,C 180,E1 -4767.692,E2 -4767.692} C_VEL
LIN {X 0,Y 523.25,Z 787.786,A -85,B 0,C 180,E1 -4769.231,E2 -4769.231} C_VEL
LIN {X 0,Y 523.246,Z 788,A -85,B 0,C 180,E1 -4770.001,E2 -4770.001} C_VEL
LIN {X 0,Y 523.274,Z 787.181,A -85,B 0,C 180,E1 -4771.54,E2 -4771.54} C_VEL
LIN {X 0,Y 523.334,Z 786.192,A -85,B 0,C 180,E1 -4772.31,E2 -4772.31} C_VEL
LIN {X 0,Y 523.368,Z 784.805,A -85,B 0,C 180,E1 -4773.08,E2 -4773.08} C_VEL
LIN {X 0,Y 523.441,Z 781.892,A -85,B 0,C 180,E1 -4774.236,E2 -4774.236} C_VEL
LIN {X 0,Y 523.464,Z 777.947,A -85,B 0,C 180,E1 -4775.393,E2 -4775.393} C_VEL
LIN {X 0,Y 523.524,Z 772.725,A -85,B 0,C 180,E1 -4776.581,E2 -4776.581} C_VEL
LIN {X 0,Y 523.666,Z 766.46,A -85,B 0,C 180,E1 -4777.713,E2 -4777.713} C_VEL
LIN {X 0,Y 523.854,Z 758.435,A -85,B 0,C 180,E1 -4778.876,E2 -4778.876} C_VEL
LIN {X 0,Y 524.08,Z 750.253,A -85,B 0,C 180,E1 -4779.845,E2 -4779.845} C_VEL
LIN {X 0,Y 524.355,Z 740.278,A -85,B 0,C 180,E1 -4780.816,E2 -4780.816} C_VEL
LIN {X 0,Y 524.665,Z 729.022,A -85,B 0,C 180,E1 -4781.689,E2 -4781.689} C_VEL
LIN {X 0,Y 524.915,Z 717.978,A -85,B 0,C 180,E1 -4782.37,E2 -4782.37} C_VEL
LIN {X 0,Y 525.154,Z 705.757,A -85,B 0,C 180,E1 -4782.954,E2 -4782.954} C_VEL
LIN {X 0,Y 525.393,Z 692.929,A -85,B 0,C 180,E1 -4783.391,E2 -4783.391} C_VEL
LIN {X 0,Y 525.573,Z 679.319,A -85,B 0,C 180,E1 -4783.682,E2 -4783.682} C_VEL
LIN {X 0,Y 525.891,Z 585.512,A -85,B 0,C 180,E1 -4784.971,E2 -4784.971} C_VEL
LIN {X 0,Y 524.35,Z 575.817,A -85,B 0,C 180,E1 -4785.166,E2 -4785.166} C_VEL
LIN {X 0,Y 524.436,Z 570.524,A -85,B 0,C 180,E1 -4785.946,E2 -4785.946} C_VEL
LIN {X 0,Y 524.84,Z 551.462,A -85,B 0,C 180,E1 -4788.95,E2 -4788.95} C_VEL
LIN {X 0,Y 525.326,Z 532.396,A -85,B 0,C 180,E1 -4792,E2 -4792} C_VEL
LIN {X 0,Y 525.463,Z 527.31,A -85,B 0,C 180,E1 -4792.823,E2 -4792.823} C_VEL
LIN {X 0,Y 523.978,Z 519.356,A -85,B 0,C 180,E1 -4794.228,E2 -4794.228} C_VEL
LIN {X 0,Y 523.956,Z 519.217,A -85,B 0,C 180,E1 -4797.133,E2 -4797.133} C_VEL
LIN {X 0,Y 523.946,Z 519.209,A -85,B 0,C 180,E1 -4799.756,E2 -4799.756} C_VEL
LIN {X 0,Y 523.938,Z 519.222,A -85,B 0,C 180,E1 -4802.45,E2 -4802.45} C_VEL
LIN {X 0,Y 523.924,Z 519.219,A -85,B 0,C 180,E1 -4805.227,E2 -4805.227} C_VEL
LIN {X 0,Y 523.92,Z 519.227,A -85,B 0,C 180,E1 -4808.102,E2 -4808.102} C_VEL
LIN {X 0,Y 523.946,Z 519.216,A -85,B 0,C 180,E1 -4811.092,E2 -4811.092} C_VEL
LIN {X 0,Y 523.944,Z 519.222,A -85,B 0,C 180,E1 -4814.228,E2 -4814.228} C_VEL
LIN {X 0,Y 523.926,Z 519.219,A -85,B 0,C 180,E1 -4816.833,E2 -4816.833} C_VEL
LIN {X 0,Y 523.949,Z 519.216,A -85,B 0,C 180,E1 -4818.908,E2 -4818.908} C_VEL
LIN {X 0,Y 523.921,Z 519.227,A -85,B 0,C 180,E1 -4821.898,E2 -4821.898} C_VEL
LIN {X 0,Y 523.943,Z 519.217,A -85,B 0,C 180,E1 -4824.909,E2 -4824.909} C_VEL
LIN {X 0,Y 523.942,Z 519.224,A -85,B 0,C 180,E1 -4827.679,E2 -4827.679} C_VEL
LIN {X 0,Y 523.958,Z 519.217,A -85,B 0,C 180,E1 -4830.677,E2 -4830.677} C_VEL
LIN {X 0,Y 524.001,Z 519.217,A -85,B 0,C 180,E1 -4833.73,E2 -4833.73} C_VEL
LIN {X 0,Y 524.065,Z 519.459,A -85,B 0,C 180,E1 -4834.075,E2 -4834.075} C_VEL
LIN {X 0,Y 525.541,Z 528.431,A -85,B 0,C 180,E1 -4835.298,E2 -4835.298} C_VEL
LIN {X 0,Y 525.284,Z 550.734,A -85,B 0,C 180,E1 -4838.205,E2 -4838.205} C_VEL
LIN {X 0,Y 524.946,Z 573.614,A -85,B 0,C 180,E1 -4841.258,E2 -4841.258} C_VEL
LIN {X 0,Y 524.675,Z 590.159,A -85,B 0,C 180,E1 -4843.462,E2 -4843.462} C_VEL
LIN {X 0,Y 524.269,Z 611.703,A -85,B 0,C 180,E1 -4846.432,E2 -4846.432} C_VEL
LIN {X 0,Y 524.049,Z 631.023,A -85,B 0,C 180,E1 -4849.032,E2 -4849.032} C_VEL
LIN {X 0,Y 524.668,Z 637.596,A -85,B 0,C 180,E1 -4849.167,E2 -4849.167} C_VEL
LIN {X 0,Y 524.516,Z 702.211,A -85,B 0,C 180,E1 -4850.066,E2 -4850.066} C_VEL
LIN {X 0,Y 524.432,Z 713.614,A -85,B 0,C 180,E1 -4850.381,E2 -4850.381} C_VEL
LIN {X 0,Y 524.295,Z 724.409,A -85,B 0,C 180,E1 -4850.841,E2 -4850.841} C_VEL
LIN {X 0,Y 524.109,Z 734.223,A -85,B 0,C 180,E1 -4851.421,E2 -4851.421} C_VEL
LIN {X 0,Y 523.871,Z 744.05,A -85,B 0,C 180,E1 -4852.193,E2 -4852.193} C_VEL
LIN {X 0,Y 523.711,Z 752.572,A -85,B 0,C 180,E1 -4853.063,E2 -4853.063} C_VEL
LIN {X 0,Y 523.654,Z 759.948,A -85,B 0,C 180,E1 -4854.03,E2 -4854.03} C_VEL
LIN {X 0,Y 523.462,Z 765.693,A -85,B 0,C 180,E1 -4854.994,E2 -4854.994} C_VEL
LIN {X 0,Y 523.467,Z 770.886,A -85,B 0,C 180,E1 -4856.151,E2 -4856.151} C_VEL
LIN {X 0,Y 523.414,Z 773.483,A -85,B 0,C 180,E1 -4856.921,E2 -4856.921} C_VEL
LIN {X 0,Y 523.338,Z 775.432,A -85,B 0,C 180,E1 -4857.691,E2 -4857.691} C_VEL
LIN {X 0,Y 523.272,Z 776.825,A -85,B 0,C 180,E1 -4858.461,E2 -4858.461} C_VEL
LIN {X 0,Y 523.246,Z 777.677,A -85,B 0,C 180,E1 -4859.23,E2 -4859.23} C_VEL
LIN {X 0,Y 523.245,Z 777.997,A -85,B 0,C 180,E1 -4860,E2 -4860} C_VEL
LIN {X 0,Y 523.248,Z 777.756,A -85,B 0,C 180,E1 -4860.77,E2 -4860.77} C_VEL
LIN {X 0,Y 523.274,Z 776.959,A -85,B 0,C 180,E1 -4861.539,E2 -4861.539} C_VEL
LIN {X 0,Y 523.334,Z 775.621,A -85,B 0,C 180,E1 -4862.309,E2 -4862.309} C_VEL
LIN {X 0,Y 523.41,Z 772.542,A -85,B 0,C 180,E1 -4863.464,E2 -4863.464} C_VEL
LIN {X 0,Y 523.439,Z 768.009,A -85,B 0,C 180,E1 -4864.621,E2 -4864.621} C_VEL
LIN {X 0,Y 523.548,Z 762.961,A -85,B 0,C 180,E1 -4865.585,E2 -4865.585} C_VEL
LIN {X 0,Y 523.692,Z 756.492,A -85,B 0,C 180,E1 -4866.544,E2 -4866.544} C_VEL
LIN {X 0,Y 523.77,Z 749.922,A -85,B 0,C 180,E1 -4867.324,E2 -4867.324} C_VEL
LIN {X 0,Y 523.93,Z 741.757,A -85,B 0,C 180,E1 -4868.097,E2 -4868.097} C_VEL
LIN {X 0,Y 524.149,Z 732.633,A -85,B 0,C 180,E1 -4868.773,E2 -4868.773} C_VEL
LIN {X 0,Y 524.304,Z 722.27,A -85,B 0,C 180,E1 -4869.354,E2 -4869.354} C_VEL
LIN {X 0,Y 524.418,Z 711.312,A -85,B 0,C 180,E1 -4869.79,E2 -4869.79} C_VEL
LIN {X 0,Y 524.532,Z 700.749,A -85,B 0,C 180,E1 -4870.055,E2 -4870.055} C_VEL
LIN {X 0,Y 524.642,Z 637.041,A -85,B 0,C 180,E1 -4870.932,E2 -4870.932} C_VEL
LIN {X 0,Y 524.072,Z 631.421,A -85,B 0,C 180,E1 -4871.041,E2 -4871.041} C_VEL
LIN {X 0,Y 524.042,Z 629.746,A -85,B 0,C 180,E1 -4871.213,E2 -4871.213} C_VEL
LIN {X 0,Y 524.429,Z 605.319,A -85,B 0,C 180,E1 -4874.553,E2 -4874.553} C_VEL
LIN {X 0,Y 524.868,Z 582.217,A -85,B 0,C 180,E1 -4877.736,E2 -4877.736} C_VEL
LIN {X 0,Y 525.276,Z 559.941,A -85,B 0,C 180,E1 -4880.78,E2 -4880.78} C_VEL
LIN {X 0,Y 525.696,Z 540.652,A -85,B 0,C 180,E1 -4883.436,E2 -4883.436} C_VEL
LIN {X 0,Y 525.763,Z 528.512,A -85,B 0,C 180,E1 -4885.112,E2 -4885.112} C_VEL
LIN {X 0,Y 524.003,Z 519.315,A -85,B 0,C 180,E1 -4886.511,E2 -4886.511} C_VEL
LIN {X 0,Y 523.949,Z 519.218,A -85,B 0,C 180,E1 -4889.528,E2 -4889.528} C_VEL
LIN {X 0,Y 523.938,Z 519.225,A -85,B 0,C 180,E1 -4892.449,E2 -4892.449} C_VEL
LIN {X 0,Y 523.925,Z 519.221,A -85,B 0,C 180,E1 -4892.875,E2 -4892.875} C_VEL
LIN {X 0,Y 523.265,Z 519.302,A -85,B 0,C 180,E1 -4893.517,E2 -4893.517} C_VEL
LIN {X 0,Y 520.409,Z 519.664,A -85,B 0,C 180,E1 -4894.559,E2 -4894.559} C_VEL
LIN {X 0,Y 517.993,Z 519.961,A -85,B 0,C 180,E1 -4895.398,E2 -4895.398} C_VEL
LIN {X 0,Y 516.96,Z 520.089,A -85,B 0,C 180,E1 -4896.046,E2 -4896.046} C_VEL
LIN {X 0,Y 516.878,Z 520.098,A -85,B 0,C 180,E1 -4896.266,E2 -4896.266} C_VEL
LIN {X 0,Y 516.891,Z 520.093,A -85,B 0,C 180,E1 -4899.194,E2 -4899.194} C_VEL
LIN {X 0,Y 516.917,Z 520.083,A -85,B 0,C 180,E1 -4901.775,E2 -4901.775} C_VEL
LIN {X 0,Y 516.928,Z 520.09,A -85,B 0,C 180,E1 -4905.01,E2 -4905.01} C_VEL
LIN {X 0,Y 516.921,Z 520.097,A -85,B 0,C 180,E1 -4908.398,E2 -4908.398} C_VEL
LIN {X 0,Y 516.886,Z 520.091,A -85,B 0,C 180,E1 -4911.284,E2 -4911.284} C_VEL
LIN {X 0,Y 516.876,Z 520.1,A -85,B 0,C 180,E1 -4914.219,E2 -4914.219} C_VEL
LIN {X 0,Y 516.9,Z 520.096,A -85,B 0,C 180,E1 -4917.053,E2 -4917.053} C_VEL
LIN {X 0,Y 516.897,Z 520.094,A -85,B 0,C 180,E1 -4919.796,E2 -4919.796} C_VEL
LIN {X 0,Y 516.931,Z 520.096,A -85,B 0,C 180,E1 -4922.467,E2 -4922.467} C_VEL
LIN {X 0,Y 516.881,Z 520.096,A -85,B 0,C 180,E1 -4925.07,E2 -4925.07} C_VEL
LIN {X 0,Y 516.874,Z 520.098,A -85,B 0,C 180,E1 -4927.621,E2 -4927.621} C_VEL
LIN {X 0,Y 516.973,Z 520.26,A -85,B 0,C 180,E1 -4929.248,E2 -4929.248} C_VEL
LIN {X 0,Y 517.793,Z 525.612,A -85,B 0,C 180,E1 -4930.37,E2 -4930.37} C_VEL
LIN {X 0,Y 517.387,Z 541.23,A -85,B 0,C 180,E1 -4933.425,E2 -4933.425} C_VEL
LIN {X 0,Y 517.249,Z 547.884,A -85,B 0,C 180,E1 -4934.662,E2 -4934.662} C_VEL
LIN {X 0,Y 518.106,Z 552.974,A -85,B 0,C 180,E1 -4934.794,E2 -4934.794} C_VEL
LIN {X 0,Y 519.111,Z 559.435,A -85,B 0,C 180,E1 -4934.916,E2 -4934.916} C_VEL
LIN {X 0,Y 518.653,Z 654.653,A -85,B 0,C 180,E1 -4936.257,E2 -4936.257} C_VEL
LIN {X 0,Y 518.469,Z 667.841,A -85,B 0,C 180,E1 -4936.602,E2 -4936.602} C_VEL
LIN {X 0,Y 518.205,Z 679.938,A -85,B 0,C 180,E1 -4937.068,E2 -4937.068} C_VEL
LIN {X 0,Y 517.96,Z 691.546,A -85,B 0,C 180,E1 -4937.673,E2 -4937.673} C_VEL
LIN {X 0,Y 517.66,Z 703.014,A -85,B 0,C 180,E1 -4938.448,E2 -4938.448} C_VEL
LIN {X 0,Y 517.306,Z 713.493,A -85,B 0,C 180,E1 -4939.332,E2 -4939.332} C_VEL
LIN {X 0,Y 517.055,Z 722.051,A -85,B 0,C 180,E1 -4940.217,E2 -4940.217} C_VEL
LIN {X 0,Y 516.835,Z 729.933,A -85,B 0,C 180,E1 -4941.2,E2 -4941.2} C_VEL
LIN {X 0,Y 516.602,Z 737.639,A -85,B 0,C 180,E1 -4942.377,E2 -4942.377} C_VEL
LIN {X 0,Y 516.45,Z 744.708,A -85,B 0,C 180,E1 -4943.749,E2 -4943.749} C_VEL
LIN {X 0,Y 516.314,Z 749.42,A -85,B 0,C 180,E1 -4944.923,E2 -4944.923} C_VEL
LIN {X 0,Y 516.373,Z 753.023,A -85,B 0,C 180,E1 -4946.097,E2 -4946.097} C_VEL
LIN {X 0,Y 516.283,Z 754.889,A -85,B 0,C 180,E1 -4946.878,E2 -4946.878} C_VEL
LIN {X 0,Y 516.261,Z 756.298,A -85,B 0,C 180,E1 -4947.659,E2 -4947.659} C_VEL
LIN {X 0,Y 516.16,Z 757.917,A -85,B 0,C 180,E1 -4949.219,E2 -4949.219} C_VEL
LIN {X 0,Y 516.155,Z 758.155,A -85,B 0,C 180,E1 -4949.999,E2 -4949.999} C_VEL
LIN {X 0,Y 516.16,Z 757.973,A -85,B 0,C 180,E1 -4950.779,E2 -4950.779} C_VEL
LIN {X 0,Y 516.261,Z 756.429,A -85,B 0,C 180,E1 -4952.34,E2 -4952.34} C_VEL
LIN {X 0,Y 516.283,Z 755.076,A -85,B 0,C 180,E1 -4953.121,E2 -4953.121} C_VEL
LIN {X 0,Y 516.361,Z 752.212,A -85,B 0,C 180,E1 -4954.292,E2 -4954.292} C_VEL
LIN {X 0,Y 516.403,Z 748.332,A -85,B 0,C 180,E1 -4955.466,E2 -4955.466} C_VEL
LIN {X 0,Y 516.481,Z 742.515,A -85,B 0,C 180,E1 -4956.808,E2 -4956.808} C_VEL
LIN {X 0,Y 516.652,Z 735.808,A -85,B 0,C 180,E1 -4958.014,E2 -4958.014} C_VEL
LIN {X 0,Y 516.88,Z 727.661,A -85,B 0,C 180,E1 -4959.192,E2 -4959.192} C_VEL
LIN {X 0,Y 517.098,Z 719.324,A -85,B 0,C 180,E1 -4960.176,E2 -4960.176} C_VEL
LIN {X 0,Y 517.475,Z 709.029,A -85,B 0,C 180,E1 -4961.158,E2 -4961.158} C_VEL
LIN {X 0,Y 517.789,Z 697.502,A -85,B 0,C 180,E1 -4962.038,E2 -4962.038} C_VEL
LIN {X 0,Y 518.082,Z 685.861,A -85,B 0,C 180,E1 -4962.734,E2 -4962.734} C_VEL
LIN {X 0,Y 518.41,Z 673.841,A -85,B 0,C 180,E1 -4963.274,E2 -4963.274} C_VEL
LIN {X 0,Y 518.534,Z 661.695,A -85,B 0,C 180,E1 -4963.67,E2 -4963.67} C_VEL
LIN {X 0,Y 518.743,Z 648.313,A -85,B 0,C 180,E1 -4963.939,E2 -4963.939} C_VEL
LIN {X 0,Y 519.026,Z 557.934,A -85,B 0,C 180,E1 -4965.198,E2 -4965.198} C_VEL
LIN {X 0,Y 517.293,Z 548.216,A -85,B 0,C 180,E1 -4965.406,E2 -4965.406} C_VEL
LIN {X 0,Y 517.24,Z 547.422,A -85,B 0,C 180,E1 -4965.485,E2 -4965.485} C_VEL
LIN {X 0,Y 517.619,Z 532.327,A -85,B 0,C 180,E1 -4968.401,E2 -4968.401} C_VEL
LIN {X 0,Y 517.715,Z 525.037,A -85,B 0,C 180,E1 -4969.838,E2 -4969.838} C_VEL
LIN {X 0,Y 516.926,Z 520.124,A -85,B 0,C 180,E1 -4970.908,E2 -4970.908} C_VEL
LIN {X 0,Y 516.904,Z 520.094,A -85,B 0,C 180,E1 -4974.362,E2 -4974.362} C_VEL
LIN {X 0,Y 516.926,Z 520.089,A -85,B 0,C 180,E1 -4976.657,E2 -4976.657} C_VEL
LIN {X 0,Y 516.911,Z 520.094,A -85,B 0,C 180,E1 -4979.523,E2 -4979.523} C_VEL
LIN {X 0,Y 516.9,Z 520.093,A -85,B 0,C 180,E1 -4982.543,E2 -4982.543} C_VEL
LIN {X 0,Y 516.881,Z 520.103,A -85,B 0,C 180,E1 -4985.331,E2 -4985.331} C_VEL
LIN {X 0,Y 516.88,Z 520.098,A -85,B 0,C 180,E1 -4987.942,E2 -4987.942} C_VEL
LIN {X 0,Y 516.883,Z 520.094,A -85,B 0,C 180,E1 -4990.74,E2 -4990.74} C_VEL
LIN {X 0,Y 516.902,Z 520.094,A -85,B 0,C 180,E1 -4992.828,E2 -4992.828} C_VEL
LIN {X 0,Y 516.919,Z 520.09,A -85,B 0,C 180,E1 -4995.009,E2 -4995.009} C_VEL
LIN {X 0,Y 516.918,Z 520.09,A -85,B 0,C 180,E1 -4998.397,E2 -4998.397} C_VEL
LIN {X 0,Y 516.902,Z 520.093,A -85,B 0,C 180,E1 -5001.286,E2 -5001.286} C_VEL
LIN {X 0,Y 516.887,Z 520.095,A -85,B 0,C 180,E1 -5004.221,E2 -5004.221} C_VEL
LIN {X 0,Y 516.893,Z 520.096,A -85,B 0,C 180,E1 -5007.053,E2 -5007.053} C_VEL
LIN {X 0,Y 516.896,Z 520.098,A -85,B 0,C 180,E1 -5009.796,E2 -5009.796} C_VEL
LIN {X 0,Y 516.924,Z 520.086,A -85,B 0,C 180,E1 -5012.467,E2 -5012.467} C_VEL
LIN {X 0,Y 516.906,Z 520.095,A -85,B 0,C 180,E1 -5015.071,E2 -5015.071} C_VEL
LIN {X 0,Y 516.88,Z 520.092,A -85,B 0,C 180,E1 -5018.462,E2 -5018.462} C_VEL
LIN {X 0,Y 516.898,Z 520.094,A -85,B 0,C 180,E1 -5020.955,E2 -5020.955} C_VEL
LIN {X 0,Y 516.911,Z 520.096,A -85,B 0,C 180,E1 -5023.41,E2 -5023.41} C_VEL
LIN {X 0,Y 516.888,Z 520.098,A -85,B 0,C 180,E1 -5025.833,E2 -5025.833} C_VEL
LIN {X 0,Y 516.957,Z 520.085,A -85,B 0,C 180,E1 -5028.233,E2 -5028.233} C_VEL
LIN {X 0,Y 516.965,Z 520.088,A -85,B 0,C 180,E1 -5031.4,E2 -5031.4} C_VEL
LIN {X 0,Y 517.003,Z 520.085,A -85,B 0,C 180,E1 -5033.757,E2 -5033.757} C_VEL
LIN {X 0,Y 517.077,Z 520.076,A -85,B 0,C 180,E1 -5037.663,E2 -5037.663} C_VEL
LIN {X 0,Y 517.088,Z 520.07,A -85,B 0,C 180,E1 -5040.779,E2 -5040.779} C_VEL
LIN {X 0,Y 517.009,Z 520.08,A -85,B 0,C 180,E1 -5043.117,E2 -5043.117} C_VEL
LIN {X 0,Y 517.003,Z 520.081,A -85,B 0,C 180,E1 -5046.243,E2 -5046.243} C_VEL
LIN {X 0,Y 516.947,Z 520.092,A -85,B 0,C 180,E1 -5049.389,E2 -5049.389} C_VEL
LIN {X 0,Y 516.976,Z 520.089,A -85,B 0,C 180,E1 -5051.824,E2 -5051.824} C_VEL
LIN {X 0,Y 516.936,Z 520.09,A -85,B 0,C 180,E1 -5055.147,E2 -5055.147} C_VEL
LIN {X 0,Y 516.919,Z 520.092,A -85,B 0,C 180,E1 -5058.222,E2 -5058.222} C_VEL
LIN {X 0,Y 516.906,Z 520.091,A -85,B 0,C 180,E1 -5060.702,E2 -5060.702} C_VEL
LIN {X 0,Y 516.904,Z 520.095,A -85,B 0,C 180,E1 -5064.072,E2 -5064.072} C_VEL
LIN {X 0,Y 516.923,Z 520.087,A -85,B 0,C 180,E1 -5066.658,E2 -5066.658} C_VEL
LIN {X 0,Y 516.905,Z 520.1,A -85,B 0,C 180,E1 -5069.525,E2 -5069.525} C_VEL
LIN {X 0,Y 516.895,Z 520.093,A -85,B 0,C 180,E1 -5072.545,E2 -5072.545} C_VEL
LIN {X 0,Y 516.879,Z 520.098,A -85,B 0,C 180,E1 -5075.333,E2 -5075.333} C_VEL
LIN {X 0,Y 516.876,Z 520.1,A -85,B 0,C 180,E1 -5077.944,E2 -5077.944} C_VEL
LIN {X 0,Y 516.881,Z 520.095,A -85,B 0,C 180,E1 -5080.742,E2 -5080.742} C_VEL
LIN {X 0,Y 516.879,Z 520.091,A -85,B 0,C 180,E1 -5082.832,E2 -5082.832} C_VEL
LIN {X 0,Y 516.918,Z 520.092,A -85,B 0,C 180,E1 -5085.011,E2 -5085.011} C_VEL
LIN {X 0,Y 516.919,Z 520.092,A -85,B 0,C 180,E1 -5088.398,E2 -5088.398} C_VEL
LIN {X 0,Y 516.884,Z 520.096,A -85,B 0,C 180,E1 -5091.286,E2 -5091.286} C_VEL
LIN {X 0,Y 516.885,Z 520.098,A -85,B 0,C 180,E1 -5094.222,E2 -5094.222} C_VEL
LIN {X 0,Y 516.896,Z 520.09,A -85,B 0,C 180,E1 -5097.054,E2 -5097.054} C_VEL
LIN {X 0,Y 516.891,Z 520.079,A -85,B 0,C 180,E1 -5099.797,E2 -5099.797} C_VEL
LIN {X 0,Y 516.928,Z 520.089,A -85,B 0,C 180,E1 -5102.468,E2 -5102.468} C_VEL
LIN {X 0,Y 516.921,Z 520.118,A -85,B 0,C 180,E1 -5105.518,E2 -5105.518} C_VEL
LIN {X 0,Y 516.936,Z 520.334,A -85,B 0,C 180,E1 -5105.63,E2 -5105.63} C_VEL
LIN {X 0,Y 518.489,Z 529.103,A -85,B 0,C 180,E1 -5107.18,E2 -5107.18} C_VEL
LIN {X 0,Y 518.038,Z 546.242,A -85,B 0,C 180,E1 -5109.973,E2 -5109.973} C_VEL
LIN {X 0,Y 517.566,Z 564,A -85,B 0,C 180,E1 -5112.823,E2 -5112.823} C_VEL
LIN {X 0,Y 517.372,Z 575.517,A -85,B 0,C 180,E1 -5114.617,E2 -5114.617} C_VEL
LIN {X 0,Y 519.067,Z 586.669,A -85,B 0,C 180,E1 -5114.846,E2 -5114.846} C_VEL
LIN {X 0,Y 518.684,Z 683.539,A -85,B 0,C 180,E1 -5116.209,E2 -5116.209} C_VEL
LIN {X 0,Y 518.431,Z 696.04,A -85,B 0,C 180,E1 -5116.527,E2 -5116.527} C_VEL
LIN {X 0,Y 518.162,Z 708.971,A -85,B 0,C 180,E1 -5117.019,E2 -5117.019} C_VEL
LIN {X 0,Y 517.871,Z 721.324,A -85,B 0,C 180,E1 -5117.663,E2 -5117.663} C_VEL
LIN {X 0,Y 517.572,Z 732.861,A -85,B 0,C 180,E1 -5118.447,E2 -5118.447} C_VEL
LIN {X 0,Y 517.222,Z 743.305,A -85,B 0,C 180,E1 -5119.332,E2 -5119.332} C_VEL
LIN {X 0,Y 516.993,Z 751.849,A -85,B 0,C 180,E1 -5120.217,E2 -5120.217} C_VEL
LIN {X 0,Y 516.773,Z 759.73,A -85,B 0,C 180,E1 -5121.2,E2 -5121.2} C_VEL
LIN {X 0,Y 516.562,Z 767.428,A -85,B 0,C 180,E1 -5122.378,E2 -5122.378} C_VEL
LIN {X 0,Y 516.424,Z 774.523,A -85,B 0,C 180,E1 -5123.75,E2 -5123.75} C_VEL
LIN {X 0,Y 516.313,Z 779.244,A -85,B 0,C 180,E1 -5124.925,E2 -5124.925} C_VEL
LIN {X 0,Y 516.354,Z 782.857,A -85,B 0,C 180,E1 -5126.099,E2 -5126.099} C_VEL
LIN {X 0,Y 516.282,Z 784.716,A -85,B 0,C 180,E1 -5126.879,E2 -5126.879} C_VEL
LIN {X 0,Y 516.26,Z 786.11,A -85,B 0,C 180,E1 -5127.66,E2 -5127.66} C_VEL
LIN {X 0,Y 516.16,Z 787.708,A -85,B 0,C 180,E1 -5129.221,E2 -5129.221} C_VEL
LIN {X 0,Y 516.154,Z 787.924,A -85,B 0,C 180,E1 -5130.001,E2 -5130.001} C_VEL
LIN {X 0,Y 516.192,Z 787.1,A -85,B 0,C 180,E1 -5131.561,E2 -5131.561} C_VEL
LIN {X 0,Y 516.26,Z 786.105,A -85,B 0,C 180,E1 -5132.341,E2 -5132.341} C_VEL
LIN {X 0,Y 516.283,Z 784.71,A -85,B 0,C 180,E1 -5133.122,E2 -5133.122} C_VEL
LIN {X 0,Y 516.327,Z 781.779,A -85,B 0,C 180,E1 -5134.294,E2 -5134.294} C_VEL
LIN {X 0,Y 516.405,Z 777.81,A -85,B 0,C 180,E1 -5135.467,E2 -5135.467} C_VEL
LIN {X 0,Y 516.465,Z 772.519,A -85,B 0,C 180,E1 -5136.679,E2 -5136.679} C_VEL
LIN {X 0,Y 516.598,Z 766.257,A -85,B 0,C 180,E1 -5137.82,E2 -5137.82} C_VEL
LIN {X 0,Y 516.811,Z 758.229,A -85,B 0,C 180,E1 -5138.998,E2 -5138.998} C_VEL
LIN {X 0,Y 517.053,Z 750.047,A -85,B 0,C 180,E1 -5139.981,E2 -5139.981} C_VEL
LIN {X 0,Y 517.334,Z 740.072,A -85,B 0,C 180,E1 -5140.965,E2 -5140.965} C_VEL
LIN {X 0,Y 517.635,Z 730.23,A -85,B 0,C 180,E1 -5141.752,E2 -5141.752} C_VEL
LIN {X 0,Y 517.923,Z 719.059,A -85,B 0,C 180,E1 -5142.468,E2 -5142.468} C_VEL
LIN {X 0,Y 518.189,Z 706.684,A -85,B 0,C 180,E1 -5143.081,E2 -5143.081} C_VEL
LIN {X 0,Y 518.474,Z 693.64,A -85,B 0,C 180,E1 -5143.548,E2 -5143.548} C_VEL
LIN {X 0,Y 518.696,Z 680.621,A -85,B 0,C 180,E1 -5143.842,E2 -5143.842} C_VEL
LIN {X 0,Y 518.988,Z 585.897,A -85,B 0,C 180,E1 -5145.167,E2 -5145.167} C_VEL
LIN {X 0,Y 517.346,Z 575.442,A -85,B 0,C 180,E1 -5145.389,E2 -5145.389} C_VEL
LIN {X 0,Y 517.816,Z 555.094,A -85,B 0,C 180,E1 -5148.6,E2 -5148.6} C_VEL
LIN {X 0,Y 518.288,Z 536.033,A -85,B 0,C 180,E1 -5151.686,E2 -5151.686} C_VEL
LIN {X 0,Y 518.525,Z 529.042,A -85,B 0,C 180,E1 -5152.829,E2 -5152.829} C_VEL
LIN {X 0,Y 516.959,Z 520.311,A -85,B 0,C 180,E1 -5154.376,E2 -5154.376} C_VEL
LIN {X 0,Y 516.93,Z 520.096,A -85,B 0,C 180,E1 -5156.658,E2 -5156.658} C_VEL
LIN {X 0,Y 516.915,Z 520.082,A -85,B 0,C 180,E1 -5159.524,E2 -5159.524} C_VEL
LIN {X 0,Y 516.9,Z 520.098,A -85,B 0,C 180,E1 -5162.544,E2 -5162.544} C_VEL
LIN {X 0,Y 516.87,Z 520.098,A -85,B 0,C 180,E1 -5165.33,E2 -5165.33} C_VEL
LIN {X 0,Y 516.885,Z 520.102,A -85,B 0,C 180,E1 -5167.943,E2 -5167.943} C_VEL
LIN {X 0,Y 516.888,Z 520.096,A -85,B 0,C 180,E1 -5170.742,E2 -5170.742} C_VEL
LIN {X 0,Y 516.888,Z 520.096,A -85,B 0,C 180,E1 -5172.831,E2 -5172.831} C_VEL
LIN {X 0,Y 516.927,Z 520.091,A -85,B 0,C 180,E1 -5175.01,E2 -5175.01} C_VEL
LIN {X 0,Y 516.921,Z 520.094,A -85,B 0,C 180,E1 -5178.398,E2 -5178.398} C_VEL
LIN {X 0,Y 516.886,Z 520.097,A -85,B 0,C 180,E1 -5181.284,E2 -5181.284} C_VEL
LIN {X 0,Y 516.895,Z 520.099,A -85,B 0,C 180,E1 -5184.221,E2 -5184.221} C_VEL
LIN {X 0,Y 516.9,Z 520.095,A -85,B 0,C 180,E1 -5187.053,E2 -5187.053} C_VEL
LIN {X 0,Y 516.896,Z 520.103,A -85,B 0,C 180,E1 -5189.796,E2 -5189.796} C_VEL
LIN {X 0,Y 516.93,Z 520.096,A -85,B 0,C 180,E1 -5192.467,E2 -5192.467} C_VEL
LIN {X 0,Y 517.026,Z 520.307,A -85,B 0,C 180,E1 -5193.945,E2 -5193.945} C_VEL
LIN {X 0,Y 518.587,Z 530.443,A -85,B 0,C 180,E1 -5195.341,E2 -5195.341} C_VEL
LIN {X 0,Y 518.257,Z 553.016,A -85,B 0,C 180,E1 -5198.313,E2 -5198.313} C_VEL
LIN {X 0,Y 517.94,Z 574.763,A -85,B 0,C 180,E1 -5201.22,E2 -5201.22} C_VEL
LIN {X 0,Y 517.642,Z 592.785,A -85,B 0,C 180,E1 -5203.637,E2 -5203.637} C_VEL
LIN {X 0,Y 517.196,Z 614.324,A -85,B 0,C 180,E1 -5206.644,E2 -5206.644} C_VEL
LIN {X 0,Y 517.022,Z 631.035,A -85,B 0,C 180,E1 -5208.883,E2 -5208.883} C_VEL
LIN {X 0,Y 517.744,Z 638.974,A -85,B 0,C 180,E1 -5209.045,E2 -5209.045} C_VEL
LIN {X 0,Y 517.517,Z 702.675,A -85,B 0,C 180,E1 -5209.955,E2 -5209.955} C_VEL
LIN {X 0,Y 517.408,Z 713.894,A -85,B 0,C 180,E1 -5210.274,E2 -5210.274} C_VEL
LIN {X 0,Y 517.267,Z 724.147,A -85,B 0,C 180,E1 -5210.715,E2 -5210.715} C_VEL
LIN {X 0,Y 517.082,Z 734.024,A -85,B 0,C 180,E1 -5211.303,E2 -5211.303} C_VEL
LIN {X 0,Y 516.858,Z 742.867,A -85,B 0,C 180,E1 -5211.988,E2 -5211.988} C_VEL
LIN {X 0,Y 516.71,Z 750.815,A -85,B 0,C 180,E1 -5212.772,E2 -5212.772} C_VEL
LIN {X 0,Y 516.622,Z 758.568,A -85,B 0,C 180,E1 -5213.752,E2 -5213.752} C_VEL
LIN {X 0,Y 516.391,Z 764.631,A -85,B 0,C 180,E1 -5214.729,E2 -5214.729} C_VEL
LIN {X 0,Y 516.417,Z 769.34,A -85,B 0,C 180,E1 -5215.707,E2 -5215.707} C_VEL
LIN {X 0,Y 516.326,Z 773.503,A -85,B 0,C 180,E1 -5216.879,E2 -5216.879} C_VEL
LIN {X 0,Y 516.266,Z 775.459,A -85,B 0,C 180,E1 -5217.659,E2 -5217.659} C_VEL
LIN {X 0,Y 516.189,Z 776.858,A -85,B 0,C 180,E1 -5218.44,E2 -5218.44} C_VEL
LIN {X 0,Y 516.156,Z 777.712,A -85,B 0,C 180,E1 -5219.22,E2 -5219.22} C_VEL
LIN {X 0,Y 516.152,Z 778.029,A -85,B 0,C 180,E1 -5220,E2 -5220} C_VEL
LIN {X 0,Y 516.158,Z 777.788,A -85,B 0,C 180,E1 -5220.78,E2 -5220.78} C_VEL
LIN {X 0,Y 516.191,Z 776.989,A -85,B 0,C 180,E1 -5221.56,E2 -5221.56} C_VEL
LIN {X 0,Y 516.261,Z 775.644,A -85,B 0,C 180,E1 -5222.341,E2 -5222.341} C_VEL
LIN {X 0,Y 516.328,Z 772.562,A -85,B 0,C 180,E1 -5223.512,E2 -5223.512} C_VEL
LIN {X 0,Y 516.343,Z 768.006,A -85,B 0,C 180,E1 -5224.684,E2 -5224.684} C_VEL
LIN {X 0,Y 516.5,Z 762.938,A -85,B 0,C 180,E1 -5225.662,E2 -5225.662} C_VEL
LIN {X 0,Y 516.627,Z 757.157,A -85,B 0,C 180,E1 -5226.538,E2 -5226.538} C_VEL
LIN {X 0,Y 516.711,Z 749.837,A -85,B 0,C 180,E1 -5227.424,E2 -5227.424} C_VEL
LIN {X 0,Y 516.893,Z 741.621,A -85,B 0,C 180,E1 -5228.208,E2 -5228.208} C_VEL
LIN {X 0,Y 517.114,Z 732.461,A -85,B 0,C 180,E1 -5228.893,E2 -5228.893} C_VEL
LIN {X 0,Y 517.298,Z 722.025,A -85,B 0,C 180,E1 -5229.482,E2 -5229.482} C_VEL
LIN {X 0,Y 517.409,Z 710.901,A -85,B 0,C 180,E1 -5229.924,E2 -5229.924} C_VEL
LIN {X 0,Y 517.544,Z 699.974,A -85,B 0,C 180,E1 -5230.193,E2 -5230.193} C_VEL
LIN {X 0,Y 517.702,Z 637.765,A -85,B 0,C 180,E1 -5231.065,E2 -5231.065} C_VEL
LIN {X 0,Y 517.085,Z 631.614,A -85,B 0,C 180,E1 -5231.188,E2 -5231.188} C_VEL
LIN {X 0,Y 517.004,Z 630.51,A -85,B 0,C 180,E1 -5231.263,E2 -5231.263} C_VEL
LIN {X 0,Y 517.394,Z 606.578,A -85,B 0,C 180,E1 -5234.554,E2 -5234.554} C_VEL
LIN {X 0,Y 517.782,Z 586.311,A -85,B 0,C 180,E1 -5237.374,E2 -5237.374} C_VEL
LIN {X 0,Y 518.238,Z 565.62,A -85,B 0,C 180,E1 -5240.232,E2 -5240.232} C_VEL
LIN {X 0,Y 518.667,Z 544.732,A -85,B 0,C 180,E1 -5243.139,E2 -5243.139} C_VEL
LIN {X 0,Y 518.917,Z 531.089,A -85,B 0,C 180,E1 -5245.018,E2 -5245.018} C_VEL
LIN {X 0,Y 516.976,Z 520.194,A -85,B 0,C 180,E1 -5246.682,E2 -5246.682} C_VEL
LIN {X 0,Y 516.915,Z 520.094,A -85,B 0,C 180,E1 -5249.524,E2 -5249.524} C_VEL
LIN {X 0,Y 516.9,Z 520.101,A -85,B 0,C 180,E1 -5252.543,E2 -5252.543} C_VEL
LIN {X 0,Y 516.888,Z 520.095,A -85,B 0,C 180,E1 -5255.332,E2 -5255.332} C_VEL
LIN {X 0,Y 516.878,Z 520.098,A -85,B 0,C 180,E1 -5256.266,E2 -5256.266} C_VEL
LIN {X 0,Y 516.22,Z 520.183,A -85,B 0,C 180,E1 -5256.916,E2 -5256.916} C_VEL
LIN {X 0,Y 513.373,Z 520.536,A -85,B 0,C 180,E1 -5257.972,E2 -5257.972} C_VEL
LIN {X 0,Y 510.958,Z 520.836,A -85,B 0,C 180,E1 -5258.823,E2 -5258.823} C_VEL
LIN {X 0,Y 509.915,Z 520.962,A -85,B 0,C 180,E1 -5259.48,E2 -5259.48} C_VEL
LIN {X 0,Y 509.828,Z 520.972,A -85,B 0,C 180,E1 -5259.702,E2 -5259.702} C_VEL
LIN {X 0,Y 509.837,Z 520.965,A -85,B 0,C 180,E1 -5262.49,E2 -5262.49} C_VEL
LIN {X 0,Y 509.862,Z 520.968,A -85,B 0,C 180,E1 -5265.332,E2 -5265.332} C_VEL
LIN {X 0,Y 509.862,Z 520.973,A -85,B 0,C 180,E1 -5268.575,E2 -5268.575} C_VEL
LIN {X 0,Y 509.856,Z 520.967,A -85,B 0,C 180,E1 -5271.786,E2 -5271.786} C_VEL
LIN {X 0,Y 509.835,Z 520.978,A -85,B 0,C 180,E1 -5274.622,E2 -5274.622} C_VEL
LIN {X 0,Y 509.866,Z 520.97,A -85,B 0,C 180,E1 -5277.481,E2 -5277.481} C_VEL
LIN {X 0,Y 509.864,Z 520.974,A -85,B 0,C 180,E1 -5280.273,E2 -5280.273} C_VEL
LIN {X 0,Y 509.889,Z 520.971,A -85,B 0,C 180,E1 -5282.944,E2 -5282.944} C_VEL
LIN {X 0,Y 509.853,Z 520.968,A -85,B 0,C 180,E1 -5285.573,E2 -5285.573} C_VEL
LIN {X 0,Y 509.934,Z 521.09,A -85,B 0,C 180,E1 -5289.076,E2 -5289.076} C_VEL
LIN {X 0,Y 510.819,Z 526.819,A -85,B 0,C 180,E1 -5290.3,E2 -5290.3} C_VEL
LIN {X 0,Y 510.406,Z 542.458,A -85,B 0,C 180,E1 -5293.398,E2 -5293.398} C_VEL
LIN {X 0,Y 510.272,Z 548.114,A -85,B 0,C 180,E1 -5294.452,E2 -5294.452} C_VEL
LIN {X 0,Y 511.943,Z 557.378,A -85,B 0,C 180,E1 -5294.666,E2 -5294.666} C_VEL
LIN {X 0,Y 512.252,Z 561.172,A -85,B 0,C 180,E1 -5294.73,E2 -5294.73} C_VEL
LIN {X 0,Y 511.778,Z 654.886,A -85,B 0,C 180,E1 -5296.069,E2 -5296.069} C_VEL
LIN {X 0,Y 511.569,Z 668.065,A -85,B 0,C 180,E1 -5296.417,E2 -5296.417} C_VEL
LIN {X 0,Y 511.3,Z 680.157,A -85,B 0,C 180,E1 -5296.891,E2 -5296.891} C_VEL
LIN {X 0,Y 511.012,Z 691.805,A -85,B 0,C 180,E1 -5297.505,E2 -5297.505} C_VEL
LIN {X 0,Y 510.71,Z 703.226,A -85,B 0,C 180,E1 -5298.288,E2 -5298.288} C_VEL
LIN {X 0,Y 510.326,Z 713.705,A -85,B 0,C 180,E1 -5299.184,E2 -5299.184} C_VEL
LIN {X 0,Y 510.058,Z 722.26,A -85,B 0,C 180,E1 -5300.082,E2 -5300.082} C_VEL
LIN {X 0,Y 509.821,Z 730.141,A -85,B 0,C 180,E1 -5301.078,E2 -5301.078} C_VEL
LIN {X 0,Y 509.56,Z 737.848,A -85,B 0,C 180,E1 -5302.271,E2 -5302.271} C_VEL
LIN {X 0,Y 509.388,Z 744.915,A -85,B 0,C 180,E1 -5303.662,E2 -5303.662} C_VEL
LIN {X 0,Y 509.248,Z 749.627,A -85,B 0,C 180,E1 -5304.853,E2 -5304.853} C_VEL
LIN {X 0,Y 509.303,Z 753.227,A -85,B 0,C 180,E1 -5306.043,E2 -5306.043} C_VEL
LIN {X 0,Y 509.202,Z 755.093,A -85,B 0,C 180,E1 -5306.835,E2 -5306.835} C_VEL
LIN {X 0,Y 509.19,Z 756.501,A -85,B 0,C 180,E1 -5307.626,E2 -5307.626} C_VEL
LIN {X 0,Y 509.074,Z 758.122,A -85,B 0,C 180,E1 -5309.208,E2 -5309.208} C_VEL
LIN {X 0,Y 509.066,Z 758.36,A -85,B 0,C 180,E1 -5309.999,E2 -5309.999} C_VEL
LIN {X 0,Y 509.073,Z 758.177,A -85,B 0,C 180,E1 -5310.79,E2 -5310.79} C_VEL
LIN {X 0,Y 509.19,Z 756.632,A -85,B 0,C 180,E1 -5312.372,E2 -5312.372} C_VEL
LIN {X 0,Y 509.202,Z 755.28,A -85,B 0,C 180,E1 -5313.164,E2 -5313.164} C_VEL
LIN {X 0,Y 509.282,Z 752.416,A -85,B 0,C 180,E1 -5314.352,E2 -5314.352} C_VEL
LIN {X 0,Y 509.345,Z 748.534,A -85,B 0,C 180,E1 -5315.542,E2 -5315.542} C_VEL
LIN {X 0,Y 509.41,Z 743.532,A -85,B 0,C 180,E1 -5316.733,E2 -5316.733} C_VEL
LIN {X 0,Y 509.595,Z 737.231,A -85,B 0,C 180,E1 -5317.926,E2 -5317.926} C_VEL
LIN {X 0,Y 509.802,Z 729.34,A -85,B 0,C 180,E1 -5319.121,E2 -5319.121} C_VEL
LIN {X 0,Y 510.103,Z 719.524,A -85,B 0,C 180,E1 -5320.317,E2 -5320.317} C_VEL
LIN {X 0,Y 510.509,Z 709.226,A -85,B 0,C 180,E1 -5321.313,E2 -5321.313} C_VEL
LIN {X 0,Y 510.834,Z 698.336,A -85,B 0,C 180,E1 -5322.159,E2 -5322.159} C_VEL
LIN {X 0,Y 511.09,Z 687.868,A -85,B 0,C 180,E1 -5322.81,E2 -5322.81} C_VEL
LIN {X 0,Y 511.406,Z 676.55,A -85,B 0,C 180,E1 -5323.358,E2 -5323.358} C_VEL
LIN {X 0,Y 511.658,Z 663.702,A -85,B 0,C 180,E1 -5323.807,E2 -5323.807} C_VEL
LIN {X 0,Y 511.847,Z 650.027,A -85,B 0,C 180,E1 -5324.105,E2 -5324.105} C_VEL
LIN {X 0,Y 512.139,Z 558.595,A -85,B 0,C 180,E1 -5325.4,E2 -5325.4} C_VEL
LIN {X 0,Y 510.31,Z 548.446,A -85,B 0,C 180,E1 -5325.62,E2 -5325.62} C_VEL
LIN {X 0,Y 510.257,Z 546.953,A -85,B 0,C 180,E1 -5325.814,E2 -5325.814} C_VEL
LIN {X 0,Y 510.701,Z 531.439,A -85,B 0,C 180,E1 -5328.867,E2 -5328.867} C_VEL
LIN {X 0,Y 510.644,Z 525.198,A -85,B 0,C 180,E1 -5330.124,E2 -5330.124} C_VEL
LIN {X 0,Y 509.881,Z 520.997,A -85,B 0,C 180,E1 -5331.079,E2 -5331.079} C_VEL
LIN {X 0,Y 509.87,Z 520.971,A -85,B 0,C 180,E1 -5334.425,E2 -5334.425} C_VEL
LIN {X 0,Y 509.885,Z 520.97,A -85,B 0,C 180,E1 -5337.055,E2 -5337.055} C_VEL
LIN {X 0,Y 509.856,Z 520.973,A -85,B 0,C 180,E1 -5339.75,E2 -5339.75} C_VEL
LIN {X 0,Y 509.875,Z 520.969,A -85,B 0,C 180,E1 -5342.774,E2 -5342.774} C_VEL
LIN {X 0,Y 509.841,Z 520.977,A -85,B 0,C 180,E1 -5345.58,E2 -5345.58} C_VEL
LIN {X 0,Y 509.848,Z 520.971,A -85,B 0,C 180,E1 -5348.337,E2 -5348.337} C_VEL
LIN {X 0,Y 509.856,Z 520.978,A -85,B 0,C 180,E1 -5351.424,E2 -5351.424} C_VEL
LIN {X 0,Y 509.853,Z 520.967,A -85,B 0,C 180,E1 -5354.667,E2 -5354.667} C_VEL
LIN {X 0,Y 509.857,Z 520.971,A -85,B 0,C 180,E1 -5358.102,E2 -5358.102} C_VEL
LIN {X 0,Y 509.872,Z 520.964,A -85,B 0,C 180,E1 -5360.65,E2 -5360.65} C_VEL
LIN {X 0,Y 509.832,Z 520.98,A -85,B 0,C 180,E1 -5363.647,E2 -5363.647} C_VEL
LIN {X 0,Y 509.858,Z 520.969,A -85,B 0,C 180,E1 -5366.539,E2 -5366.539} C_VEL
LIN {X 0,Y 509.845,Z 520.978,A -85,B 0,C 180,E1 -5369.334,E2 -5369.334} C_VEL
LIN {X 0,Y 509.89,Z 520.964,A -85,B 0,C 180,E1 -5372.054,E2 -5372.054} C_VEL
LIN {X 0,Y 509.872,Z 520.968,A -85,B 0,C 180,E1 -5374.704,E2 -5374.704} C_VEL
LIN {X 0,Y 509.849,Z 520.976,A -85,B 0,C 180,E1 -5377.449,E2 -5377.449} C_VEL
LIN {X 0,Y 509.91,Z 520.967,A -85,B 0,C 180,E1 -5379.844,E2 -5379.844} C_VEL
LIN {X 0,Y 509.881,Z 520.969,A -85,B 0,C 180,E1 -5383.174,E2 -5383.174} C_VEL
LIN {X 0,Y 509.857,Z 520.977,A -85,B 0,C 180,E1 -5385.634,E2 -5385.634} C_VEL
LIN {X 0,Y 509.906,Z 520.964,A -85,B 0,C 180,E1 -5388.874,E2 -5388.874} C_VEL
LIN {X 0,Y 509.945,Z 520.961,A -85,B 0,C 180,E1 -5392.078,E2 -5392.078} C_VEL
LIN {X 0,Y 509.976,Z 520.955,A -85,B 0,C 180,E1 -5394.464,E2 -5394.464} C_VEL
LIN {X 0,Y 510.048,Z 520.951,A -85,B 0,C 180,E1 -5397.631,E2 -5397.631} C_VEL
LIN {X 0,Y 510.058,Z 520.945,A -85,B 0,C 180,E1 -5400.789,E2 -5400.789} C_VEL
LIN {X 0,Y 509.952,Z 520.959,A -85,B 0,C 180,E1 -5403.16,E2 -5403.16} C_VEL
LIN {X 0,Y 509.971,Z 520.956,A -85,B 0,C 180,E1 -5406.33,E2 -5406.33} C_VEL
LIN {X 0,Y 509.909,Z 520.962,A -85,B 0,C 180,E1 -5408.72,E2 -5408.72} C_VEL
LIN {X 0,Y 509.943,Z 520.963,A -85,B 0,C 180,E1 -5411.931,E2 -5411.931} C_VEL
LIN {X 0,Y 509.886,Z 520.969,A -85,B 0,C 180,E1 -5415.242,E2 -5415.242} C_VEL
LIN {X 0,Y 509.881,Z 520.97,A -85,B 0,C 180,E1 -5418.001,E2 -5418.001} C_VEL
LIN {X 0,Y 509.844,Z 520.972,A -85,B 0,C 180,E1 -5421.002,E2 -5421.002} C_VEL
LIN {X 0,Y 509.83,Z 520.98,A -85,B 0,C 180,E1 -5423.564,E2 -5423.564} C_VEL
LIN {X 0,Y 509.907,Z 520.961,A -85,B 0,C 180,E1 -5426.38,E2 -5426.38} C_VEL
LIN {X 0,Y 509.871,Z 520.969,A -85,B 0,C 180,E1 -5428.845,E2 -5428.845} C_VEL
LIN {X 0,Y 509.82,Z 520.981,A -85,B 0,C 180,E1 -5431.59,E2 -5431.59} C_VEL
LIN {X 0,Y 509.849,Z 520.97,A -85,B 0,C 180,E1 -5434.414,E2 -5434.414} C_VEL
LIN {X 0,Y 509.814,Z 520.972,A -85,B 0,C 180,E1 -5437.341,E2 -5437.341} C_VEL
LIN {X 0,Y 509.833,Z 520.974,A -85,B 0,C 180,E1 -5440.383,E2 -5440.383} C_VEL
LIN {X 0,Y 509.818,Z 520.972,A -85,B 0,C 180,E1 -5443.063,E2 -5443.063} C_VEL
LIN {X 0,Y 509.827,Z 520.979,A -85,B 0,C 180,E1 -5445.793,E2 -5445.793} C_VEL
LIN {X 0,Y 509.862,Z 520.97,A -85,B 0,C 180,E1 -5448.576,E2 -5448.576} C_VEL
LIN {X 0,Y 509.849,Z 520.968,A -85,B 0,C 180,E1 -5451.787,E2 -5451.787} C_VEL
LIN {X 0,Y 509.84,Z 520.973,A -85,B 0,C 180,E1 -5454.624,E2 -5454.624} C_VEL
LIN {X 0,Y 509.864,Z 520.959,A -85,B 0,C 180,E1 -5457.482,E2 -5457.482} C_VEL
LIN {X 0,Y 509.857,Z 520.965,A -85,B 0,C 180,E1 -5460.275,E2 -5460.275} C_VEL
LIN {X 0,Y 509.885,Z 520.966,A -85,B 0,C 180,E1 -5462.945,E2 -5462.945} C_VEL
LIN {X 0,Y 509.878,Z 521.07,A -85,B 0,C 180,E1 -5465.399,E2 -5465.399} C_VEL
LIN {X 0,Y 511.388,Z 528.789,A -85,B 0,C 180,E1 -5466.822,E2 -5466.822} C_VEL
LIN {X 0,Y 511.386,Z 535.866,A -85,B 0,C 180,E1 -5468.008,E2 -5468.008} C_VEL
LIN {X 0,Y 510.907,Z 551.117,A -85,B 0,C 180,E1 -5470.515,E2 -5470.515} C_VEL
LIN {X 0,Y 510.459,Z 568.899,A -85,B 0,C 180,E1 -5473.401,E2 -5473.401} C_VEL
LIN {X 0,Y 510.355,Z 575.132,A -85,B 0,C 180,E1 -5474.386,E2 -5474.386} C_VEL
LIN {X 0,Y 510.95,Z 579.333,A -85,B 0,C 180,E1 -5474.498,E2 -5474.498} C_VEL
LIN {X 0,Y 512.26,Z 589.029,A -85,B 0,C 180,E1 -5474.676,E2 -5474.676} C_VEL
LIN {X 0,Y 511.807,Z 683.334,A -85,B 0,C 180,E1 -5476.02,E2 -5476.02} C_VEL
LIN {X 0,Y 511.529,Z 695.835,A -85,B 0,C 180,E1 -5476.342,E2 -5476.342} C_VEL
LIN {X 0,Y 511.255,Z 708.767,A -85,B 0,C 180,E1 -5476.84,E2 -5476.84} C_VEL
LIN {X 0,Y 510.918,Z 721.175,A -85,B 0,C 180,E1 -5477.496,E2 -5477.496} C_VEL
LIN {X 0,Y 510.59,Z 732.655,A -85,B 0,C 180,E1 -5478.287,E2 -5478.287} C_VEL
LIN {X 0,Y 510.24,Z 743.1,A -85,B 0,C 180,E1 -5479.184,E2 -5479.184} C_VEL
LIN {X 0,Y 509.971,Z 751.643,A -85,B 0,C 180,E1 -5480.081,E2 -5480.081} C_VEL
LIN {X 0,Y 509.712,Z 759.523,A -85,B 0,C 180,E1 -5481.077,E2 -5481.077} C_VEL
LIN {X 0,Y 509.512,Z 767.223,A -85,B 0,C 180,E1 -5482.272,E2 -5482.272} C_VEL
LIN {X 0,Y 509.325,Z 774.318,A -85,B 0,C 180,E1 -5483.663,E2 -5483.663} C_VEL
LIN {X 0,Y 509.248,Z 779.039,A -85,B 0,C 180,E1 -5484.854,E2 -5484.854} C_VEL
LIN {X 0,Y 509.25,Z 782.651,A -85,B 0,C 180,E1 -5486.044,E2 -5486.044} C_VEL
LIN {X 0,Y 509.2,Z 784.512,A -85,B 0,C 180,E1 -5486.836,E2 -5486.836} C_VEL
LIN {X 0,Y 509.189,Z 785.906,A -85,B 0,C 180,E1 -5487.628,E2 -5487.628} C_VEL
LIN {X 0,Y 509.073,Z 787.504,A -85,B 0,C 180,E1 -5489.21,E2 -5489.21} C_VEL
LIN {X 0,Y 509.065,Z 787.719,A -85,B 0,C 180,E1 -5490.001,E2 -5490.001} C_VEL
LIN {X 0,Y 509.112,Z 786.895,A -85,B 0,C 180,E1 -5491.583,E2 -5491.583} C_VEL
LIN {X 0,Y 509.189,Z 785.901,A -85,B 0,C 180,E1 -5492.374,E2 -5492.374} C_VEL
LIN {X 0,Y 509.201,Z 784.505,A -85,B 0,C 180,E1 -5493.165,E2 -5493.165} C_VEL
LIN {X 0,Y 509.216,Z 781.573,A -85,B 0,C 180,E1 -5494.354,E2 -5494.354} C_VEL
LIN {X 0,Y 509.322,Z 777.604,A -85,B 0,C 180,E1 -5495.544,E2 -5495.544} C_VEL
LIN {X 0,Y 509.402,Z 771.946,A -85,B 0,C 180,E1 -5496.845,E2 -5496.845} C_VEL
LIN {X 0,Y 509.573,Z 764.815,A -85,B 0,C 180,E1 -5498.128,E2 -5498.128} C_VEL
LIN {X 0,Y 509.794,Z 756.531,A -85,B 0,C 180,E1 -5499.323,E2 -5499.323} C_VEL
LIN {X 0,Y 510.05,Z 748.04,A -85,B 0,C 180,E1 -5500.32,E2 -5500.32} C_VEL
LIN {X 0,Y 510.432,Z 737.552,A -85,B 0,C 180,E1 -5501.316,E2 -5501.316} C_VEL
LIN {X 0,Y 510.716,Z 726.895,A -85,B 0,C 180,E1 -5502.134,E2 -5502.134} C_VEL
LIN {X 0,Y 511.068,Z 715.799,A -85,B 0,C 180,E1 -5502.812,E2 -5502.812} C_VEL
LIN {X 0,Y 511.368,Z 704.138,A -85,B 0,C 180,E1 -5503.36,E2 -5503.36} C_VEL
LIN {X 0,Y 511.629,Z 690.687,A -85,B 0,C 180,E1 -5503.809,E2 -5503.809} C_VEL
LIN {X 0,Y 511.85,Z 677.391,A -85,B 0,C 180,E1 -5504.081,E2 -5504.081} C_VEL
LIN {X 0,Y 512.122,Z 586.638,A -85,B 0,C 180,E1 -5505.362,E2 -5505.362} C_VEL
LIN {X 0,Y 510.374,Z 575.47,A -85,B 0,C 180,E1 -5505.59,E2 -5505.59} C_VEL
LIN {X 0,Y 510.412,Z 571.397,A -85,B 0,C 180,E1 -5506.191,E2 -5506.191} C_VEL
LIN {X 0,Y 510.884,Z 553.65,A -85,B 0,C 180,E1 -5509.07,E2 -5509.07} C_VEL
LIN {X 0,Y 511.44,Z 534.587,A -85,B 0,C 180,E1 -5512.204,E2 -5512.204} C_VEL
LIN {X 0,Y 511.384,Z 528.77,A -85,B 0,C 180,E1 -5513.182,E2 -5513.182} C_VEL
LIN {X 0,Y 509.924,Z 521.23,A -85,B 0,C 180,E1 -5514.544,E2 -5514.544} C_VEL
LIN {X 0,Y 509.882,Z 520.965,A -85,B 0,C 180,E1 -5515.296,E2 -5515.296} C_VEL
LIN {X 0,Y 509.895,Z 520.963,A -85,B 0,C 180,E1 -5518.1,E2 -5518.1} C_VEL
LIN {X 0,Y 509.85,Z 520.973,A -85,B 0,C 180,E1 -5521.28,E2 -5521.28} C_VEL
LIN {X 0,Y 509.86,Z 520.978,A -85,B 0,C 180,E1 -5524.203,E2 -5524.203} C_VEL
LIN {X 0,Y 509.821,Z 520.976,A -85,B 0,C 180,E1 -5527.341,E2 -5527.341} C_VEL
LIN {X 0,Y 509.842,Z 520.977,A -85,B 0,C 180,E1 -5530.382,E2 -5530.382} C_VEL
LIN {X 0,Y 509.828,Z 520.975,A -85,B 0,C 180,E1 -5533.063,E2 -5533.063} C_VEL
LIN {X 0,Y 509.835,Z 520.981,A -85,B 0,C 180,E1 -5535.792,E2 -5535.792} C_VEL
LIN {X 0,Y 509.863,Z 520.972,A -85,B 0,C 180,E1 -5538.575,E2 -5538.575} C_VEL
LIN {X 0,Y 509.856,Z 520.979,A -85,B 0,C 180,E1 -5541.786,E2 -5541.786} C_VEL
LIN {X 0,Y 509.85,Z 520.973,A -85,B 0,C 180,E1 -5544.623,E2 -5544.623} C_VEL
LIN {X 0,Y 509.867,Z 520.975,A -85,B 0,C 180,E1 -5547.481,E2 -5547.481} C_VEL
LIN {X 0,Y 509.862,Z 520.976,A -85,B 0,C 180,E1 -5550.274,E2 -5550.274} C_VEL
LIN {X 0,Y 509.893,Z 520.972,A -85,B 0,C 180,E1 -5552.945,E2 -5552.945} C_VEL
LIN {X 0,Y 509.952,Z 521.165,A -85,B 0,C 180,E1 -5553.799,E2 -5553.799} C_VEL
LIN {X 0,Y 511.549,Z 530.106,A -85,B 0,C 180,E1 -5555.061,E2 -5555.061} C_VEL
LIN {X 0,Y 511.331,Z 549.094,A -85,B 0,C 180,E1 -5557.579,E2 -5557.579} C_VEL
LIN {X 0,Y 511.044,Z 569.442,A -85,B 0,C 180,E1 -5560.31,E2 -5560.31} C_VEL
LIN {X 0,Y 510.679,Z 590.97,A -85,B 0,C 180,E1 -5563.202,E2 -5563.202} C_VEL
LIN {X 0,Y 510.212,Z 612.655,A -85,B 0,C 180,E1 -5566.254,E2 -5566.254} C_VEL
LIN {X 0,Y 510.009,Z 631.239,A -85,B 0,C 180,E1 -5568.745,E2 -5568.745} C_VEL
LIN {X 0,Y 510.779,Z 640.425,A -85,B 0,C 180,E1 -5568.919,E2 -5568.919} C_VEL
LIN {X 0,Y 510.537,Z 702.011,A -85,B 0,C 180,E1 -5569.816,E2 -5569.816} C_VEL
LIN {X 0,Y 510.432,Z 712.75,A -85,B 0,C 180,E1 -5570.115,E2 -5570.115} C_VEL
LIN {X 0,Y 510.274,Z 722.886,A -85,B 0,C 180,E1 -5570.537,E2 -5570.537} C_VEL
LIN {X 0,Y 510.061,Z 733.825,A -85,B 0,C 180,E1 -5571.182,E2 -5571.182} C_VEL
LIN {X 0,Y 509.821,Z 742.723,A -85,B 0,C 180,E1 -5571.877,E2 -5571.877} C_VEL
LIN {X 0,Y 509.659,Z 750.745,A -85,B 0,C 180,E1 -5572.672,E2 -5572.672} C_VEL
LIN {X 0,Y 509.555,Z 758.524,A -85,B 0,C 180,E1 -5573.665,E2 -5573.665} C_VEL
LIN {X 0,Y 509.331,Z 764.631,A -85,B 0,C 180,E1 -5574.656,E2 -5574.656} C_VEL
LIN {X 0,Y 509.343,Z 769.363,A -85,B 0,C 180,E1 -5575.648,E2 -5575.648} C_VEL
LIN {X 0,Y 509.241,Z 773.524,A -85,B 0,C 180,E1 -5576.835,E2 -5576.835} C_VEL
LIN {X 0,Y 509.196,Z 775.498,A -85,B 0,C 180,E1 -5577.627,E2 -5577.627} C_VEL
LIN {X 0,Y 509.11,Z 776.913,A -85,B 0,C 180,E1 -5578.418,E2 -5578.418} C_VEL
LIN {X 0,Y 509.07,Z 777.773,A -85,B 0,C 180,E1 -5579.209,E2 -5579.209} C_VEL
LIN {X 0,Y 509.064,Z 778.084,A -85,B 0,C 180,E1 -5580,E2 -5580} C_VEL
LIN {X 0,Y 509.072,Z 777.841,A -85,B 0,C 180,E1 -5580.791,E2 -5580.791} C_VEL
LIN {X 0,Y 509.112,Z 777.041,A -85,B 0,C 180,E1 -5581.582,E2 -5581.582} C_VEL
LIN {X 0,Y 509.191,Z 775.679,A -85,B 0,C 180,E1 -5582.373,E2 -5582.373} C_VEL
LIN {X 0,Y 509.25,Z 772.594,A -85,B 0,C 180,E1 -5583.561,E2 -5583.561} C_VEL
LIN {X 0,Y 509.252,Z 768.004,A -85,B 0,C 180,E1 -5584.75,E2 -5584.75} C_VEL
LIN {X 0,Y 509.447,Z 762.905,A -85,B 0,C 180,E1 -5585.74,E2 -5585.74} C_VEL
LIN {X 0,Y 509.557,Z 756.172,A -85,B 0,C 180,E1 -5586.756,E2 -5586.756} C_VEL
LIN {X 0,Y 509.694,Z 747.846,A -85,B 0,C 180,E1 -5587.726,E2 -5587.726} C_VEL
LIN {X 0,Y 509.941,Z 739.12,A -85,B 0,C 180,E1 -5588.52,E2 -5588.52} C_VEL
LIN {X 0,Y 510.178,Z 729.111,A -85,B 0,C 180,E1 -5589.215,E2 -5589.215} C_VEL
LIN {X 0,Y 510.323,Z 718.475,A -85,B 0,C 180,E1 -5589.763,E2 -5589.763} C_VEL
LIN {X 0,Y 510.497,Z 707.108,A -85,B 0,C 180,E1 -5590.16,E2 -5590.16} C_VEL
LIN {X 0,Y 510.581,Z 695.996,A -85,B 0,C 180,E1 -5590.383,E2 -5590.383} C_VEL
LIN {X 0,Y 510.661,Z 637.508,A -85,B 0,C 180,E1 -5591.22,E2 -5591.22} C_VEL
LIN {X 0,Y 509.975,Z 631.001,A -85,B 0,C 180,E1 -5591.366,E2 -5591.366} C_VEL
LIN {X 0,Y 510.373,Z 607.912,A -85,B 0,C 180,E1 -5594.555,E2 -5594.555} C_VEL
LIN {X 0,Y 510.853,Z 584.694,A -85,B 0,C 180,E1 -5597.801,E2 -5597.801} C_VEL
LIN {X 0,Y 511.325,Z 563.922,A -85,B 0,C 180,E1 -5600.708,E2 -5600.708} C_VEL
LIN {X 0,Y 511.788,Z 544.222,A -85,B 0,C 180,E1 -5603.468,E2 -5603.468} C_VEL
LIN {X 0,Y 511.974,Z 531.947,A -85,B 0,C 180,E1 -5605.185,E2 -5605.185} C_VEL
LIN {X 0,Y 509.93,Z 521.071,A -85,B 0,C 180,E1 -5606.861,E2 -5606.861} C_VEL
LIN {X 0,Y 509.861,Z 520.974,A -85,B 0,C 180,E1 -5609.751,E2 -5609.751} C_VEL
LIN {X 0,Y 509.877,Z 520.973,A -85,B 0,C 180,E1 -5612.774,E2 -5612.774} C_VEL
LIN {X 0,Y 509.848,Z 520.972,A -85,B 0,C 180,E1 -5615.581,E2 -5615.581} C_VEL
LIN {X 0,Y 509.855,Z 520.978,A -85,B 0,C 180,E1 -5618.338,E2 -5618.338} C_VEL
LIN {X 0,Y 509.828,Z 520.972,A -85,B 0,C 180,E1 -5619.702,E2 -5619.702} C_VEL
LIN {X 0,Y 509.148,Z 521.063,A -85,B 0,C 180,E1 -5620.361,E2 -5620.361} C_VEL
LIN {X 0,Y 506.275,Z 521.409,A -85,B 0,C 180,E1 -5621.431,E2 -5621.431} C_VEL
LIN {X 0,Y 503.863,Z 521.71,A -85,B 0,C 180,E1 -5622.293,E2 -5622.293} C_VEL
LIN {X 0,Y 502.847,Z 521.834,A -85,B 0,C 180,E1 -5622.959,E2 -5622.959} C_VEL
LIN {X 0,Y 502.774,Z 521.841,A -85,B 0,C 180,E1 -5623.184,E2 -5623.184} C_VEL
LIN {X 0,Y 502.795,Z 521.848,A -85,B 0,C 180,E1 -5625.661,E2 -5625.661} C_VEL
LIN {X 0,Y 502.835,Z 521.846,A -85,B 0,C 180,E1 -5627.864,E2 -5627.864} C_VEL
LIN {X 0,Y 502.807,Z 521.847,A -85,B 0,C 180,E1 -5631.024,E2 -5631.024} C_VEL
LIN {X 0,Y 502.779,Z 521.856,A -85,B 0,C 180,E1 -5634.169,E2 -5634.169} C_VEL
LIN {X 0,Y 502.837,Z 521.849,A -85,B 0,C 180,E1 -5636.993,E2 -5636.993} C_VEL
LIN {X 0,Y 502.82,Z 521.85,A -85,B 0,C 180,E1 -5640.065,E2 -5640.065} C_VEL
LIN {X 0,Y 502.838,Z 521.852,A -85,B 0,C 180,E1 -5642.533,E2 -5642.533} C_VEL
LIN {X 0,Y 502.791,Z 521.848,A -85,B 0,C 180,E1 -5645.309,E2 -5645.309} C_VEL
LIN {X 0,Y 502.787,Z 521.853,A -85,B 0,C 180,E1 -5647.826,E2 -5647.826} C_VEL
LIN {X 0,Y 502.891,Z 522.016,A -85,B 0,C 180,E1 -5648.931,E2 -5648.931} C_VEL
LIN {X 0,Y 503.862,Z 528.027,A -85,B 0,C 180,E1 -5650.229,E2 -5650.229} C_VEL
LIN {X 0,Y 503.455,Z 542.644,A -85,B 0,C 180,E1 -5653.162,E2 -5653.162} C_VEL
LIN {X 0,Y 503.288,Z 548.253,A -85,B 0,C 180,E1 -5654.227,E2 -5654.227} C_VEL
LIN {X 0,Y 504.598,Z 555.475,A -85,B 0,C 180,E1 -5654.406,E2 -5654.406} C_VEL
LIN {X 0,Y 505.432,Z 560.209,A -85,B 0,C 180,E1 -5654.502,E2 -5654.502} C_VEL
LIN {X 0,Y 504.918,Z 655.119,A -85,B 0,C 180,E1 -5655.875,E2 -5655.875} C_VEL
LIN {X 0,Y 504.696,Z 668.288,A -85,B 0,C 180,E1 -5656.229,E2 -5656.229} C_VEL
LIN {X 0,Y 504.403,Z 680.375,A -85,B 0,C 180,E1 -5656.708,E2 -5656.708} C_VEL
LIN {X 0,Y 504.089,Z 692.228,A -85,B 0,C 180,E1 -5657.344,E2 -5657.344} C_VEL
LIN {X 0,Y 503.769,Z 703.439,A -85,B 0,C 180,E1 -5658.125,E2 -5658.125} C_VEL
LIN {X 0,Y 503.359,Z 713.916,A -85,B 0,C 180,E1 -5659.033,E2 -5659.033} C_VEL
LIN {X 0,Y 503.068,Z 722.471,A -85,B 0,C 180,E1 -5659.942,E2 -5659.942} C_VEL
LIN {X 0,Y 502.804,Z 730.351,A -85,B 0,C 180,E1 -5660.952,E2 -5660.952} C_VEL
LIN {X 0,Y 502.52,Z 738.056,A -85,B 0,C 180,E1 -5662.162,E2 -5662.162} C_VEL
LIN {X 0,Y 502.325,Z 745.123,A -85,B 0,C 180,E1 -5663.573,E2 -5663.573} C_VEL
LIN {X 0,Y 502.186,Z 749.833,A -85,B 0,C 180,E1 -5664.78,E2 -5664.78} C_VEL
LIN {X 0,Y 502.235,Z 753.433,A -85,B 0,C 180,E1 -5665.987,E2 -5665.987} C_VEL
LIN {X 0,Y 502.124,Z 755.298,A -85,B 0,C 180,E1 -5666.79,E2 -5666.79} C_VEL
LIN {X 0,Y 502.121,Z 756.705,A -85,B 0,C 180,E1 -5667.593,E2 -5667.593} C_VEL
LIN {X 0,Y 501.991,Z 758.326,A -85,B 0,C 180,E1 -5669.197,E2 -5669.197} C_VEL
LIN {X 0,Y 501.98,Z 758.564,A -85,B 0,C 180,E1 -5669.999,E2 -5669.999} C_VEL
LIN {X 0,Y 501.99,Z 758.381,A -85,B 0,C 180,E1 -5670.801,E2 -5670.801} C_VEL
LIN {X 0,Y 502.121,Z 756.835,A -85,B 0,C 180,E1 -5672.406,E2 -5672.406} C_VEL
LIN {X 0,Y 502.124,Z 755.483,A -85,B 0,C 180,E1 -5673.209,E2 -5673.209} C_VEL
LIN {X 0,Y 502.205,Z 752.619,A -85,B 0,C 180,E1 -5674.414,E2 -5674.414} C_VEL
LIN {X 0,Y 502.288,Z 748.736,A -85,B 0,C 180,E1 -5675.62,E2 -5675.62} C_VEL
LIN {X 0,Y 502.351,Z 743.734,A -85,B 0,C 180,E1 -5676.828,E2 -5676.828} C_VEL
LIN {X 0,Y 502.557,Z 737.432,A -85,B 0,C 180,E1 -5678.038,E2 -5678.038} C_VEL
LIN {X 0,Y 502.782,Z 729.541,A -85,B 0,C 180,E1 -5679.25,E2 -5679.25} C_VEL
LIN {X 0,Y 503.063,Z 721.497,A -85,B 0,C 180,E1 -5680.26,E2 -5680.26} C_VEL
LIN {X 0,Y 503.464,Z 711.675,A -85,B 0,C 180,E1 -5681.269,E2 -5681.269} C_VEL
LIN {X 0,Y 503.856,Z 700.539,A -85,B 0,C 180,E1 -5682.186,E2 -5682.186} C_VEL
LIN {X 0,Y 504.119,Z 689.824,A -85,B 0,C 180,E1 -5682.888,E2 -5682.888} C_VEL
LIN {X 0,Y 504.487,Z 677.868,A -85,B 0,C 180,E1 -5683.493,E2 -5683.493} C_VEL
LIN {X 0,Y 504.773,Z 664.797,A -85,B 0,C 180,E1 -5683.973,E2 -5683.973} C_VEL
LIN {X 0,Y 505.004,Z 651.695,A -85,B 0,C 180,E1 -5684.275,E2 -5684.275} C_VEL
LIN {X 0,Y 505.316,Z 559.491,A -85,B 0,C 180,E1 -5685.603,E2 -5685.603} C_VEL
LIN {X 0,Y 503.3,Z 548.315,A -85,B 0,C 180,E1 -5685.857,E2 -5685.857} C_VEL
LIN {X 0,Y 503.468,Z 542.058,A -85,B 0,C 180,E1 -5687.045,E2 -5687.045} C_VEL
LIN {X 0,Y 503.859,Z 528.475,A -85,B 0,C 180,E1 -5689.769,E2 -5689.769} C_VEL
LIN {X 0,Y 502.869,Z 521.896,A -85,B 0,C 180,E1 -5691.213,E2 -5691.213} C_VEL
LIN {X 0,Y 502.829,Z 521.85,A -85,B 0,C 180,E1 -5694.79,E2 -5694.79} C_VEL
LIN {X 0,Y 502.834,Z 521.853,A -85,B 0,C 180,E1 -5697.466,E2 -5697.466} C_VEL
LIN {X 0,Y 502.809,Z 521.847,A -85,B 0,C 180,E1 -5700.21,E2 -5700.21} C_VEL
LIN {X 0,Y 502.831,Z 521.849,A -85,B 0,C 180,E1 -5703.03,E2 -5703.03} C_VEL
LIN {X 0,Y 502.781,Z 521.852,A -85,B 0,C 180,E1 -5705.949,E2 -5705.949} C_VEL
LIN {X 0,Y 502.8,Z 521.852,A -85,B 0,C 180,E1 -5708.975,E2 -5708.975} C_VEL
LIN {X 0,Y 502.826,Z 521.847,A -85,B 0,C 180,E1 -5712.135,E2 -5712.135} C_VEL
LIN {X 0,Y 502.797,Z 521.852,A -85,B 0,C 180,E1 -5715.467,E2 -5715.467} C_VEL
LIN {X 0,Y 502.822,Z 521.849,A -85,B 0,C 180,E1 -5719.003,E2 -5719.003} C_VEL
LIN {X 0,Y 502.792,Z 521.846,A -85,B 0,C 180,E1 -5722.046,E2 -5722.046} C_VEL
LIN {X 0,Y 502.805,Z 521.852,A -85,B 0,C 180,E1 -5725.034,E2 -5725.034} C_VEL
LIN {X 0,Y 502.783,Z 521.853,A -85,B 0,C 180,E1 -5727.915,E2 -5727.915} C_VEL
LIN {X 0,Y 502.833,Z 521.846,A -85,B 0,C 180,E1 -5730.713,E2 -5730.713} C_VEL
LIN {X 0,Y 502.875,Z 521.845,A -85,B 0,C 180,E1 -5733.434,E2 -5733.434} C_VEL
LIN {X 0,Y 502.785,Z 521.851,A -85,B 0,C 180,E1 -5736.086,E2 -5736.086} C_VEL
LIN {X 0,Y 502.777,Z 521.849,A -85,B 0,C 180,E1 -5738.688,E2 -5738.688} C_VEL
LIN {X 0,Y 502.824,Z 521.851,A -85,B 0,C 180,E1 -5741.248,E2 -5741.248} C_VEL
LIN {X 0,Y 502.817,Z 521.849,A -85,B 0,C 180,E1 -5743.767,E2 -5743.767} C_VEL
LIN {X 0,Y 502.824,Z 521.846,A -85,B 0,C 180,E1 -5746.254,E2 -5746.254} C_VEL
LIN {X 0,Y 502.87,Z 521.839,A -85,B 0,C 180,E1 -5748.717,E2 -5748.717} C_VEL
LIN {X 0,Y 502.895,Z 521.84,A -85,B 0,C 180,E1 -5751.966,E2 -5751.966} C_VEL
LIN {X 0,Y 502.932,Z 521.832,A -85,B 0,C 180,E1 -5754.386,E2 -5754.386} C_VEL
LIN {X 0,Y 503.018,Z 521.826,A -85,B 0,C 180,E1 -5757.598,E2 -5757.598} C_VEL
LIN {X 0,Y 503.019,Z 521.825,A -85,B 0,C 180,E1 -5760,E2 -5760} C_VEL
LIN {X 0,Y 503.018,Z 521.82,A -85,B 0,C 180,E1 -5762.402,E2 -5762.402} C_VEL
LIN {X 0,Y 502.932,Z 521.84,A -85,B 0,C 180,E1 -5765.614,E2 -5765.614} C_VEL
LIN {X 0,Y 502.894,Z 521.839,A -85,B 0,C 180,E1 -5768.033,E2 -5768.033} C_VEL
LIN {X 0,Y 502.885,Z 521.839,A -85,B 0,C 180,E1 -5771.283,E2 -5771.283} C_VEL
LIN {X 0,Y 502.837,Z 521.843,A -85,B 0,C 180,E1 -5774.571,E2 -5774.571} C_VEL
LIN {X 0,Y 502.855,Z 521.847,A -85,B 0,C 180,E1 -5777.907,E2 -5777.907} C_VEL
LIN {X 0,Y 502.821,Z 521.845,A -85,B 0,C 180,E1 -5780.537,E2 -5780.537} C_VEL
LIN {X 0,Y 502.79,Z 521.85,A -85,B 0,C 180,E1 -5783.041,E2 -5783.041} C_VEL
LIN {X 0,Y 502.835,Z 521.85,A -85,B 0,C 180,E1 -5785.676,E2 -5785.676} C_VEL
LIN {X 0,Y 502.834,Z 521.846,A -85,B 0,C 180,E1 -5788.373,E2 -5788.373} C_VEL
LIN {X 0,Y 502.79,Z 521.855,A -85,B 0,C 180,E1 -5791.5,E2 -5791.5} C_VEL
LIN {X 0,Y 502.802,Z 521.848,A -85,B 0,C 180,E1 -5794.446,E2 -5794.446} C_VEL
LIN {X 0,Y 502.776,Z 521.847,A -85,B 0,C 180,E1 -5797.179,E2 -5797.179} C_VEL
LIN {X 0,Y 502.783,Z 521.855,A -85,B 0,C 180,E1 -5800.016,E2 -5800.016} C_VEL
LIN {X 0,Y 502.797,Z 521.847,A -85,B 0,C 180,E1 -5802.2,E2 -5802.2} C_VEL
LIN {X 0,Y 502.797,Z 521.856,A -85,B 0,C 180,E1 -5805.469,E2 -5805.469} C_VEL
LIN {X 0,Y 502.832,Z 521.852,A -85,B 0,C 180,E1 -5807.866,E2 -5807.866} C_VEL
LIN {X 0,Y 502.807,Z 521.847,A -85,B 0,C 180,E1 -5811.026,E2 -5811.026} C_VEL
LIN {X 0,Y 502.78,Z 521.856,A -85,B 0,C 180,E1 -5814.168,E2 -5814.168} C_VEL
LIN {X 0,Y 502.831,Z 521.841,A -85,B 0,C 180,E1 -5816.994,E2 -5816.994} C_VEL
LIN {X 0,Y 502.813,Z 521.834,A -85,B 0,C 180,E1 -5820.066,E2 -5820.066} C_VEL
LIN {X 0,Y 502.834,Z 521.844,A -85,B 0,C 180,E1 -5822.534,E2 -5822.534} C_VEL
LIN {X 0,Y 502.875,Z 521.938,A -85,B 0,C 180,E1 -5825.213,E2 -5825.213} C_VEL
LIN {X 0,Y 504.222,Z 529.089,A -85,B 0,C 180,E1 -5826.555,E2 -5826.555} C_VEL
LIN {X 0,Y 504.589,Z 533.149,A -85,B 0,C 180,E1 -5827.264,E2 -5827.264} C_VEL
LIN {X 0,Y 504.033,Z 549.671,A -85,B 0,C 180,E1 -5830.026,E2 -5830.026} C_VEL
LIN {X 0,Y 503.488,Z 567.438,A -85,B 0,C 180,E1 -5832.955,E2 -5832.955} C_VEL
LIN {X 0,Y 503.327,Z 574.957,A -85,B 0,C 180,E1 -5834.164,E2 -5834.164} C_VEL
LIN {X 0,Y 504.236,Z 580.86,A -85,B 0,C 180,E1 -5834.312,E2 -5834.312} C_VEL
LIN {X 0,Y 505.407,Z 589.848,A -85,B 0,C 180,E1 -5834.478,E2 -5834.478} C_VEL
LIN {X 0,Y 504.927,Z 683.13,A -85,B 0,C 180,E1 -5835.826,E2 -5835.826} C_VEL
LIN {X 0,Y 504.634,Z 695.631,A -85,B 0,C 180,E1 -5836.152,E2 -5836.152} C_VEL
LIN {X 0,Y 504.327,Z 708.561,A -85,B 0,C 180,E1 -5836.656,E2 -5836.656} C_VEL
LIN {X 0,Y 504.001,Z 720.376,A -85,B 0,C 180,E1 -5837.284,E2 -5837.284} C_VEL
LIN {X 0,Y 503.627,Z 731.154,A -85,B 0,C 180,E1 -5838.02,E2 -5838.02} C_VEL
LIN {X 0,Y 503.287,Z 741.821,A -85,B 0,C 180,E1 -5838.931,E2 -5838.931} C_VEL
LIN {X 0,Y 502.941,Z 751.437,A -85,B 0,C 180,E1 -5839.941,E2 -5839.941} C_VEL
LIN {X 0,Y 502.672,Z 759.318,A -85,B 0,C 180,E1 -5840.951,E2 -5840.951} C_VEL
LIN {X 0,Y 502.431,Z 767.017,A -85,B 0,C 180,E1 -5842.162,E2 -5842.162} C_VEL
LIN {X 0,Y 502.234,Z 774.112,A -85,B 0,C 180,E1 -5843.573,E2 -5843.573} C_VEL
LIN {X 0,Y 502.182,Z 778.834,A -85,B 0,C 180,E1 -5844.782,E2 -5844.782} C_VEL
LIN {X 0,Y 502.144,Z 782.446,A -85,B 0,C 180,E1 -5845.988,E2 -5845.988} C_VEL
LIN {X 0,Y 502.12,Z 784.307,A -85,B 0,C 180,E1 -5846.791,E2 -5846.791} C_VEL
LIN {X 0,Y 502.091,Z 785.702,A -85,B 0,C 180,E1 -5847.594,E2 -5847.594} C_VEL
LIN {X 0,Y 501.99,Z 787.3,A -85,B 0,C 180,E1 -5849.199,E2 -5849.199} C_VEL
LIN {X 0,Y 501.98,Z 787.515,A -85,B 0,C 180,E1 -5850.001,E2 -5850.001} C_VEL
LIN {X 0,Y 502.036,Z 786.691,A -85,B 0,C 180,E1 -5851.605,E2 -5851.605} C_VEL
LIN {X 0,Y 502.091,Z 785.697,A -85,B 0,C 180,E1 -5852.407,E2 -5852.407} C_VEL
LIN {X 0,Y 502.121,Z 784.301,A -85,B 0,C 180,E1 -5853.21,E2 -5853.21} C_VEL
LIN {X 0,Y 502.112,Z 781.367,A -85,B 0,C 180,E1 -5854.416,E2 -5854.416} C_VEL
LIN {X 0,Y 502.242,Z 777.399,A -85,B 0,C 180,E1 -5855.622,E2 -5855.622} C_VEL
LIN {X 0,Y 502.333,Z 771.388,A -85,B 0,C 180,E1 -5857.012,E2 -5857.012} C_VEL
LIN {X 0,Y 502.502,Z 764.609,A -85,B 0,C 180,E1 -5858.243,E2 -5858.243} C_VEL
LIN {X 0,Y 502.759,Z 756.325,A -85,B 0,C 180,E1 -5859.454,E2 -5859.454} C_VEL
LIN {X 0,Y 503.033,Z 747.834,A -85,B 0,C 180,E1 -5860.465,E2 -5860.465} C_VEL
LIN {X 0,Y 503.447,Z 737.346,A -85,B 0,C 180,E1 -5861.475,E2 -5861.475} C_VEL
LIN {X 0,Y 503.73,Z 726.689,A -85,B 0,C 180,E1 -5862.305,E2 -5862.305} C_VEL
LIN {X 0,Y 504.122,Z 715.593,A -85,B 0,C 180,E1 -5862.992,E2 -5862.992} C_VEL
LIN {X 0,Y 504.452,Z 703.933,A -85,B 0,C 180,E1 -5863.547,E2 -5863.547} C_VEL
LIN {X 0,Y 504.721,Z 691.399,A -85,B 0,C 180,E1 -5863.976,E2 -5863.976} C_VEL
LIN {X 0,Y 504.941,Z 678.706,A -85,B 0,C 180,E1 -5864.252,E2 -5864.252} C_VEL
LIN {X 0,Y 505.313,Z 587.524,A -85,B 0,C 180,E1 -5865.558,E2 -5865.558} C_VEL
LIN {X 0,Y 503.344,Z 575.226,A -85,B 0,C 180,E1 -5865.816,E2 -5865.816} C_VEL
LIN {X 0,Y 503.428,Z 569.93,A -85,B 0,C 180,E1 -5866.63,E2 -5866.63} C_VEL
LIN {X 0,Y 503.877,Z 553.471,A -85,B 0,C 180,E1 -5869.346,E2 -5869.346} C_VEL
LIN {X 0,Y 504.51,Z 535.683,A -85,B 0,C 180,E1 -5872.31,E2 -5872.31} C_VEL
LIN {X 0,Y 504.532,Z 530.639,A -85,B 0,C 180,E1 -5873.166,E2 -5873.166} C_VEL
LIN {X 0,Y 502.875,Z 522.169,A -85,B 0,C 180,E1 -5874.712,E2 -5874.712} C_VEL
LIN {X 0,Y 502.843,Z 521.843,A -85,B 0,C 180,E1 -5875.011,E2 -5875.011} C_VEL
LIN {X 0,Y 502.835,Z 521.85,A -85,B 0,C 180,E1 -5877.467,E2 -5877.467} C_VEL
LIN {X 0,Y 502.814,Z 521.849,A -85,B 0,C 180,E1 -5880.211,E2 -5880.211} C_VEL
LIN {X 0,Y 502.836,Z 521.847,A -85,B 0,C 180,E1 -5883.032,E2 -5883.032} C_VEL
LIN {X 0,Y 502.777,Z 521.859,A -85,B 0,C 180,E1 -5885.951,E2 -5885.951} C_VEL
LIN {X 0,Y 502.805,Z 521.849,A -85,B 0,C 180,E1 -5888.976,E2 -5888.976} C_VEL
LIN {X 0,Y 502.801,Z 521.856,A -85,B 0,C 180,E1 -5892.139,E2 -5892.139} C_VEL
LIN {X 0,Y 502.805,Z 521.853,A -85,B 0,C 180,E1 -5895.468,E2 -5895.468} C_VEL
LIN {X 0,Y 502.825,Z 521.848,A -85,B 0,C 180,E1 -5898.934,E2 -5898.934} C_VEL
LIN {X 0,Y 502.798,Z 521.857,A -85,B 0,C 180,E1 -5902.046,E2 -5902.046} C_VEL
LIN {X 0,Y 502.814,Z 521.849,A -85,B 0,C 180,E1 -5905.035,E2 -5905.035} C_VEL
LIN {X 0,Y 502.789,Z 521.859,A -85,B 0,C 180,E1 -5907.916,E2 -5907.916} C_VEL
LIN {X 0,Y 502.828,Z 521.85,A -85,B 0,C 180,E1 -5910.712,E2 -5910.712} C_VEL
LIN {X 0,Y 502.938,Z 522.001,A -85,B 0,C 180,E1 -5913.644,E2 -5913.644} C_VEL
LIN {X 0,Y 504.661,Z 532.771,A -85,B 0,C 180,E1 -5915.166,E2 -5915.166} C_VEL
LIN {X 0,Y 504.305,Z 554.756,A -85,B 0,C 180,E1 -5918.112,E2 -5918.112} C_VEL
LIN {X 0,Y 503.936,Z 576.596,A -85,B 0,C 180,E1 -5921.08,E2 -5921.08} C_VEL
LIN {X 0,Y 503.493,Z 599.208,A -85,B 0,C 180,E1 -5924.167,E2 -5924.167} C_VEL
LIN {X 0,Y 503.129,Z 618.611,A -85,B 0,C 180,E1 -5926.88,E2 -5926.88} C_VEL
LIN {X 0,Y 502.955,Z 631.155,A -85,B 0,C 180,E1 -5928.58,E2 -5928.58} C_VEL
LIN {X 0,Y 503.811,Z 640.204,A -85,B 0,C 180,E1 -5928.763,E2 -5928.763} C_VEL
LIN {X 0,Y 503.52,Z 702.467,A -85,B 0,C 180,E1 -5929.698,E2 -5929.698} C_VEL
LIN {X 0,Y 503.426,Z 713.014,A -85,B 0,C 180,E1 -5930.001,E2 -5930.001} C_VEL
LIN {X 0,Y 503.235,Z 723.624,A -85,B 0,C 180,E1 -5930.454,E2 -5930.454} C_VEL
LIN {X 0,Y 503.032,Z 733.625,A -85,B 0,C 180,E1 -5931.058,E2 -5931.058} C_VEL
LIN {X 0,Y 502.762,Z 742.577,A -85,B 0,C 180,E1 -5931.762,E2 -5931.762} C_VEL
LIN {X 0,Y 502.61,Z 750.672,A -85,B 0,C 180,E1 -5932.568,E2 -5932.568} C_VEL
LIN {X 0,Y 502.475,Z 758.474,A -85,B 0,C 180,E1 -5933.576,E2 -5933.576} C_VEL
LIN {X 0,Y 502.276,Z 764.628,A -85,B 0,C 180,E1 -5934.58,E2 -5934.58} C_VEL
LIN {X 0,Y 502.251,Z 769.385,A -85,B 0,C 180,E1 -5935.586,E2 -5935.586} C_VEL
LIN {X 0,Y 502.161,Z 773.545,A -85,B 0,C 180,E1 -5936.791,E2 -5936.791} C_VEL
LIN {X 0,Y 502.099,Z 775.538,A -85,B 0,C 180,E1 -5937.593,E2 -5937.593} C_VEL
LIN {X 0,Y 502.034,Z 776.969,A -85,B 0,C 180,E1 -5938.396,E2 -5938.396} C_VEL
LIN {X 0,Y 501.987,Z 777.832,A -85,B 0,C 180,E1 -5939.198,E2 -5939.198} C_VEL
LIN {X 0,Y 501.978,Z 778.138,A -85,B 0,C 180,E1 -5940,E2 -5940} C_VEL
LIN {X 0,Y 501.989,Z 777.889,A -85,B 0,C 180,E1 -5940.802,E2 -5940.802} C_VEL
LIN {X 0,Y 502.036,Z 777.085,A -85,B 0,C 180,E1 -5941.604,E2 -5941.604} C_VEL
LIN {X 0,Y 502.093,Z 775.715,A -85,B 0,C 180,E1 -5942.407,E2 -5942.407} C_VEL
LIN {X 0,Y 502.175,Z 772.625,A -85,B 0,C 180,E1 -5943.611,E2 -5943.611} C_VEL
LIN {X 0,Y 502.168,Z 768.002,A -85,B 0,C 180,E1 -5944.817,E2 -5944.817} C_VEL
LIN {X 0,Y 502.372,Z 762.872,A -85,B 0,C 180,E1 -5945.821,E2 -5945.821} C_VEL
LIN {X 0,Y 502.503,Z 756.67,A -85,B 0,C 180,E1 -5946.779,E2 -5946.779} C_VEL
LIN {X 0,Y 502.603,Z 749.666,A -85,B 0,C 180,E1 -5947.634,E2 -5947.634} C_VEL
LIN {X 0,Y 502.835,Z 741.339,A -85,B 0,C 180,E1 -5948.439,E2 -5948.439} C_VEL
LIN {X 0,Y 503.078,Z 732.117,A -85,B 0,C 180,E1 -5949.144,E2 -5949.144} C_VEL
LIN {X 0,Y 503.289,Z 721.447,A -85,B 0,C 180,E1 -5949.748,E2 -5949.748} C_VEL
LIN {X 0,Y 503.409,Z 710.796,A -85,B 0,C 180,E1 -5950.177,E2 -5950.177} C_VEL
LIN {X 0,Y 503.568,Z 698.345,A -85,B 0,C 180,E1 -5950.479,E2 -5950.479} C_VEL
LIN {X 0,Y 503.76,Z 638.633,A -85,B 0,C 180,E1 -5951.355,E2 -5951.355} C_VEL
LIN {X 0,Y 502.943,Z 631.065,A -85,B 0,C 180,E1 -5951.519,E2 -5951.519} C_VEL
LIN {X 0,Y 503.391,Z 607.841,A -85,B 0,C 180,E1 -5954.761,E2 -5954.761} C_VEL
LIN {X 0,Y 503.943,Z 583.518,A -85,B 0,C 180,E1 -5958.184,E2 -5958.184} C_VEL
LIN {X 0,Y 504.455,Z 561.951,A -85,B 0,C 180,E1 -5961.237,E2 -5961.237} C_VEL
LIN {X 0,Y 505.019,Z 540.648,A -85,B 0,C 180,E1 -5964.238,E2 -5964.238} C_VEL
LIN {X 0,Y 505.014,Z 532.931,A -85,B 0,C 180,E1 -5965.341,E2 -5965.341} C_VEL
LIN {X 0,Y 502.877,Z 521.953,A -85,B 0,C 180,E1 -5967.042,E2 -5967.042} C_VEL
LIN {X 0,Y 502.813,Z 521.856,A -85,B 0,C 180,E1 -5970.211,E2 -5970.211} C_VEL
LIN {X 0,Y 502.836,Z 521.848,A -85,B 0,C 180,E1 -5973.031,E2 -5973.031} C_VEL
LIN {X 0,Y 502.789,Z 521.854,A -85,B 0,C 180,E1 -5975.95,E2 -5975.95} C_VEL
LIN {X 0,Y 502.807,Z 521.85,A -85,B 0,C 180,E1 -5978.976,E2 -5978.976} C_VEL
LIN {X 0,Y 502.8,Z 521.844,A -85,B 0,C 180,E1 -5982.139,E2 -5982.139} C_VEL
LIN {X 0,Y 502.774,Z 521.841,A -85,B 0,C 180,E1 -5983.184,E2 -5983.184} C_VEL
LIN {X 0,Y 502.131,Z 521.926,A -85,B 0,C 180,E1 -5983.852,E2 -5983.852} C_VEL
LIN {X 0,Y 499.276,Z 522.29,A -85,B 0,C 180,E1 -5984.938,E2 -5984.938} C_VEL
LIN {X 0,Y 496.849,Z 522.594,A -85,B 0,C 180,E1 -5985.812,E2 -5985.812} C_VEL
LIN {X 0,Y 495.809,Z 522.727,A -85,B 0,C 180,E1 -5986.488,E2 -5986.488} C_VEL
LIN {X 0,Y 495.727,Z 522.732,A -85,B 0,C 180,E1 -5986.716,E2 -5986.716} C_VEL
LIN {X 0,Y 495.771,Z 522.719,A -85,B 0,C 180,E1 -5989.3,E2 -5989.3} C_VEL
LIN {X 0,Y 495.734,Z 522.732,A -85,B 0,C 180,E1 -5992.438,E2 -5992.438} C_VEL
LIN {X 0,Y 495.782,Z 522.72,A -85,B 0,C 180,E1 -5995.457,E2 -5995.457} C_VEL
LIN {X 0,Y 495.76,Z 522.732,A -85,B 0,C 180,E1 -5998.364,E2 -5998.364} C_VEL
LIN {X 0,Y 495.793,Z 522.723,A -85,B 0,C 180,E1 -6001.507,E2 -6001.507} C_VEL
LIN {X 0,Y 495.786,Z 522.725,A -85,B 0,C 180,E1 -6003.931,E2 -6003.931} C_VEL
LIN {X 0,Y 495.754,Z 522.73,A -85,B 0,C 180,E1 -6007.495,E2 -6007.495} C_VEL
LIN {X 0,Y 495.807,Z 522.868,A -85,B 0,C 180,E1 -6008.755,E2 -6008.755} C_VEL
LIN {X 0,Y 496.889,Z 529.235,A -85,B 0,C 180,E1 -6010.156,E2 -6010.156} C_VEL
LIN {X 0,Y 496.465,Z 543.868,A -85,B 0,C 180,E1 -6013.129,E2 -6013.129} C_VEL
LIN {X 0,Y 496.324,Z 548.457,A -85,B 0,C 180,E1 -6014.001,E2 -6014.001} C_VEL
LIN {X 0,Y 497.909,Z 557.167,A -85,B 0,C 180,E1 -6014.213,E2 -6014.213} C_VEL
LIN {X 0,Y 498.599,Z 562.122,A -85,B 0,C 180,E1 -6014.308,E2 -6014.308} C_VEL
LIN {X 0,Y 498.062,Z 655.352,A -85,B 0,C 180,E1 -6015.677,E2 -6015.677} C_VEL
LIN {X 0,Y 497.797,Z 668.513,A -85,B 0,C 180,E1 -6016.034,E2 -6016.034} C_VEL
LIN {X 0,Y 497.509,Z 680.594,A -85,B 0,C 180,E1 -6016.521,E2 -6016.521} C_VEL
LIN {X 0,Y 497.184,Z 691.371,A -85,B 0,C 180,E1 -6017.099,E2 -6017.099} C_VEL
LIN {X 0,Y 496.854,Z 702.365,A -85,B 0,C 180,E1 -6017.853,E2 -6017.853} C_VEL
LIN {X 0,Y 496.411,Z 713.063,A -85,B 0,C 180,E1 -6018.774,E2 -6018.774} C_VEL
LIN {X 0,Y 496.083,Z 722.681,A -85,B 0,C 180,E1 -6019.799,E2 -6019.799} C_VEL
LIN {X 0,Y 495.77,Z 730.561,A -85,B 0,C 180,E1 -6020.823,E2 -6020.823} C_VEL
LIN {X 0,Y 495.495,Z 738.264,A -85,B 0,C 180,E1 -6022.05,E2 -6022.05} C_VEL
LIN {X 0,Y 495.253,Z 745.331,A -85,B 0,C 180,E1 -6023.481,E2 -6023.481} C_VEL
LIN {X 0,Y 495.128,Z 750.04,A -85,B 0,C 180,E1 -6024.706,E2 -6024.706} C_VEL
LIN {X 0,Y 495.15,Z 753.639,A -85,B 0,C 180,E1 -6025.93,E2 -6025.93} C_VEL
LIN {X 0,Y 495.051,Z 755.504,A -85,B 0,C 180,E1 -6026.744,E2 -6026.744} C_VEL
LIN {X 0,Y 495.025,Z 756.91,A -85,B 0,C 180,E1 -6027.558,E2 -6027.558} C_VEL
LIN {X 0,Y 494.911,Z 758.531,A -85,B 0,C 180,E1 -6029.186,E2 -6029.186} C_VEL
LIN {X 0,Y 494.898,Z 758.768,A -85,B 0,C 180,E1 -6029.999,E2 -6029.999} C_VEL
LIN {X 0,Y 494.911,Z 758.585,A -85,B 0,C 180,E1 -6030.813,E2 -6030.813} C_VEL
LIN {X 0,Y 495.025,Z 757.039,A -85,B 0,C 180,E1 -6032.44,E2 -6032.44} C_VEL
LIN {X 0,Y 495.051,Z 755.686,A -85,B 0,C 180,E1 -6033.255,E2 -6033.255} C_VEL
LIN {X 0,Y 495.114,Z 752.822,A -85,B 0,C 180,E1 -6034.477,E2 -6034.477} C_VEL
LIN {X 0,Y 495.234,Z 748.938,A -85,B 0,C 180,E1 -6035.7,E2 -6035.7} C_VEL
LIN {X 0,Y 495.304,Z 743.936,A -85,B 0,C 180,E1 -6036.926,E2 -6036.926} C_VEL
LIN {X 0,Y 495.518,Z 737.633,A -85,B 0,C 180,E1 -6038.153,E2 -6038.153} C_VEL
LIN {X 0,Y 495.776,Z 729.741,A -85,B 0,C 180,E1 -6039.381,E2 -6039.381} C_VEL
LIN {X 0,Y 496.065,Z 721.696,A -85,B 0,C 180,E1 -6040.406,E2 -6040.406} C_VEL
LIN {X 0,Y 496.509,Z 711.873,A -85,B 0,C 180,E1 -6041.429,E2 -6041.429} C_VEL
LIN {X 0,Y 496.872,Z 702.216,A -85,B 0,C 180,E1 -6042.249,E2 -6042.249} C_VEL
LIN {X 0,Y 497.152,Z 691.558,A -85,B 0,C 180,E1 -6042.981,E2 -6042.981} C_VEL
LIN {X 0,Y 497.553,Z 679.186,A -85,B 0,C 180,E1 -6043.633,E2 -6043.633} C_VEL
LIN {X 0,Y 497.881,Z 665.84,A -85,B 0,C 180,E1 -6044.144,E2 -6044.144} C_VEL
LIN {X 0,Y 498.094,Z 653.365,A -85,B 0,C 180,E1 -6044.451,E2 -6044.451} C_VEL
LIN {X 0,Y 498.543,Z 560.699,A -85,B 0,C 180,E1 -6045.805,E2 -6045.805} C_VEL
LIN {X 0,Y 496.328,Z 548.56,A -85,B 0,C 180,E1 -6046.082,E2 -6046.082} C_VEL
LIN {X 0,Y 496.367,Z 545.372,A -85,B 0,C 180,E1 -6046.661,E2 -6046.661} C_VEL
LIN {X 0,Y 496.848,Z 530.721,A -85,B 0,C 180,E1 -6049.629,E2 -6049.629} C_VEL
LIN {X 0,Y 496.313,Z 525.535,A -85,B 0,C 180,E1 -6050.732,E2 -6050.732} C_VEL
LIN {X 0,Y 495.787,Z 522.779,A -85,B 0,C 180,E1 -6051.38,E2 -6051.38} C_VEL
LIN {X 0,Y 495.753,Z 522.73,A -85,B 0,C 180,E1 -6054.274,E2 -6054.274} C_VEL
LIN {X 0,Y 495.814,Z 522.721,A -85,B 0,C 180,E1 -6056.973,E2 -6056.973} C_VEL
LIN {X 0,Y 495.764,Z 522.725,A -85,B 0,C 180,E1 -6060.146,E2 -6060.146} C_VEL
LIN {X 0,Y 495.792,Z 522.727,A -85,B 0,C 180,E1 -6063.244,E2 -6063.244} C_VEL
LIN {X 0,Y 495.726,Z 522.73,A -85,B 0,C 180,E1 -6066.089,E2 -6066.089} C_VEL
LIN {X 0,Y 495.762,Z 522.727,A -85,B 0,C 180,E1 -6068.768,E2 -6068.768} C_VEL
LIN {X 0,Y 495.774,Z 522.729,A -85,B 0,C 180,E1 -6071.778,E2 -6071.778} C_VEL
LIN {X 0,Y 495.745,Z 522.727,A -85,B 0,C 180,E1 -6075.138,E2 -6075.138} C_VEL
LIN {X 0,Y 495.756,Z 522.727,A -85,B 0,C 180,E1 -6078.219,E2 -6078.219} C_VEL
LIN {X 0,Y 495.774,Z 522.723,A -85,B 0,C 180,E1 -6081.229,E2 -6081.229} C_VEL
LIN {X 0,Y 495.753,Z 522.727,A -85,B 0,C 180,E1 -6084.463,E2 -6084.463} C_VEL
LIN {X 0,Y 495.764,Z 522.731,A -85,B 0,C 180,E1 -6087.405,E2 -6087.405} C_VEL
LIN {X 0,Y 495.776,Z 522.725,A -85,B 0,C 180,E1 -6090.254,E2 -6090.254} C_VEL
LIN {X 0,Y 495.827,Z 522.719,A -85,B 0,C 180,E1 -6093.248,E2 -6093.248} C_VEL
LIN {X 0,Y 495.746,Z 522.732,A -85,B 0,C 180,E1 -6095.725,E2 -6095.725} C_VEL
LIN {X 0,Y 495.741,Z 522.725,A -85,B 0,C 180,E1 -6098.371,E2 -6098.371} C_VEL
LIN {X 0,Y 495.778,Z 522.726,A -85,B 0,C 180,E1 -6100.971,E2 -6100.971} C_VEL
LIN {X 0,Y 495.774,Z 522.727,A -85,B 0,C 180,E1 -6103.53,E2 -6103.53} C_VEL
LIN {X 0,Y 495.787,Z 522.725,A -85,B 0,C 180,E1 -6106.055,E2 -6106.055} C_VEL
LIN {X 0,Y 495.844,Z 522.714,A -85,B 0,C 180,E1 -6108.555,E2 -6108.555} C_VEL
LIN {X 0,Y 495.866,Z 522.717,A -85,B 0,C 180,E1 -6111.852,E2 -6111.852} C_VEL
LIN {X 0,Y 495.889,Z 522.71,A -85,B 0,C 180,E1 -6114.306,E2 -6114.306} C_VEL
LIN {X 0,Y 495.987,Z 522.701,A -85,B 0,C 180,E1 -6117.564,E2 -6117.564} C_VEL
LIN {X 0,Y 495.99,Z 522.7,A -85,B 0,C 180,E1 -6120,E2 -6120} C_VEL
LIN {X 0,Y 495.987,Z 522.695,A -85,B 0,C 180,E1 -6122.436,E2 -6122.436} C_VEL
LIN {X 0,Y 495.889,Z 522.717,A -85,B 0,C 180,E1 -6125.694,E2 -6125.694} C_VEL
LIN {X 0,Y 495.865,Z 522.713,A -85,B 0,C 180,E1 -6128.148,E2 -6128.148} C_VEL
LIN {X 0,Y 495.86,Z 522.716,A -85,B 0,C 180,E1 -6131.445,E2 -6131.445} C_VEL
LIN {X 0,Y 495.782,Z 522.722,A -85,B 0,C 180,E1 -6134.783,E2 -6134.783} C_VEL
LIN {X 0,Y 495.781,Z 522.725,A -85,B 0,C 180,E1 -6137.319,E2 -6137.319} C_VEL
LIN {X 0,Y 495.771,Z 522.728,A -85,B 0,C 180,E1 -6139.89,E2 -6139.89} C_VEL
LIN {X 0,Y 495.758,Z 522.725,A -85,B 0,C 180,E1 -6142.863,E2 -6142.863} C_VEL
LIN {X 0,Y 495.793,Z 522.722,A -85,B 0,C 180,E1 -6146.068,E2 -6146.068} C_VEL
LIN {X 0,Y 495.765,Z 522.726,A -85,B 0,C 180,E1 -6148.815,E2 -6148.815} C_VEL
LIN {X 0,Y 495.753,Z 522.734,A -85,B 0,C 180,E1 -6151.727,E2 -6151.727} C_VEL
LIN {X 0,Y 495.772,Z 522.723,A -85,B 0,C 180,E1 -6154.696,E2 -6154.696} C_VEL
LIN {X 0,Y 495.726,Z 522.729,A -85,B 0,C 180,E1 -6157.562,E2 -6157.562} C_VEL
LIN {X 0,Y 495.762,Z 522.726,A -85,B 0,C 180,E1 -6160.701,E2 -6160.701} C_VEL
LIN {X 0,Y 495.729,Z 522.735,A -85,B 0,C 180,E1 -6164.002,E2 -6164.002} C_VEL
LIN {X 0,Y 495.759,Z 522.725,A -85,B 0,C 180,E1 -6167.122,E2 -6167.122} C_VEL
LIN {X 0,Y 495.78,Z 522.722,A -85,B 0,C 180,E1 -6170.366,E2 -6170.366} C_VEL
LIN {X 0,Y 495.73,Z 522.728,A -85,B 0,C 180,E1 -6173.457,E2 -6173.457} C_VEL
LIN {X 0,Y 495.758,Z 522.722,A -85,B 0,C 180,E1 -6176.437,E2 -6176.437} C_VEL
LIN {X 0,Y 495.751,Z 522.699,A -85,B 0,C 180,E1 -6179.314,E2 -6179.314} C_VEL
LIN {X 0,Y 495.781,Z 522.726,A -85,B 0,C 180,E1 -6182.11,E2 -6182.11} C_VEL
LIN {X 0,Y 495.826,Z 522.818,A -85,B 0,C 180,E1 -6185.022,E2 -6185.022} C_VEL
LIN {X 0,Y 497.677,Z 532.975,A -85,B 0,C 180,E1 -6186.93,E2 -6186.93} C_VEL
LIN {X 0,Y 497.13,Z 549.497,A -85,B 0,C 180,E1 -6189.736,E2 -6189.736} C_VEL
LIN {X 0,Y 496.487,Z 568.503,A -85,B 0,C 180,E1 -6192.92,E2 -6192.92} C_VEL
LIN {X 0,Y 496.328,Z 574.826,A -85,B 0,C 180,E1 -6193.94,E2 -6193.94} C_VEL
LIN {X 0,Y 497.721,Z 583.766,A -85,B 0,C 180,E1 -6194.146,E2 -6194.146} C_VEL
LIN {X 0,Y 498.57,Z 590.097,A -85,B 0,C 180,E1 -6194.267,E2 -6194.267} C_VEL
LIN {X 0,Y 498.064,Z 682.925,A -85,B 0,C 180,E1 -6195.626,E2 -6195.626} C_VEL
LIN {X 0,Y 497.747,Z 695.426,A -85,B 0,C 180,E1 -6195.956,E2 -6195.956} C_VEL
LIN {X 0,Y 497.416,Z 708.357,A -85,B 0,C 180,E1 -6196.467,E2 -6196.467} C_VEL
LIN {X 0,Y 497.039,Z 720.483,A -85,B 0,C 180,E1 -6197.123,E2 -6197.123} C_VEL
LIN {X 0,Y 496.618,Z 732.244,A -85,B 0,C 180,E1 -6197.952,E2 -6197.952} C_VEL
LIN {X 0,Y 496.254,Z 742.689,A -85,B 0,C 180,E1 -6198.875,E2 -6198.875} C_VEL
LIN {X 0,Y 495.894,Z 751.231,A -85,B 0,C 180,E1 -6199.797,E2 -6199.797} C_VEL
LIN {X 0,Y 495.632,Z 759.112,A -85,B 0,C 180,E1 -6200.822,E2 -6200.822} C_VEL
LIN {X 0,Y 495.375,Z 766.812,A -85,B 0,C 180,E1 -6202.05,E2 -6202.05} C_VEL
LIN {X 0,Y 495.163,Z 773.907,A -85,B 0,C 180,E1 -6203.481,E2 -6203.481} C_VEL
LIN {X 0,Y 495.118,Z 778.63,A -85,B 0,C 180,E1 -6204.707,E2 -6204.707} C_VEL
LIN {X 0,Y 495.038,Z 782.24,A -85,B 0,C 180,E1 -6205.93,E2 -6205.93} C_VEL
LIN {X 0,Y 495.042,Z 784.103,A -85,B 0,C 180,E1 -6206.745,E2 -6206.745} C_VEL
LIN {X 0,Y 494.997,Z 785.497,A -85,B 0,C 180,E1 -6207.56,E2 -6207.56} C_VEL
LIN {X 0,Y 494.962,Z 786.49,A -85,B 0,C 180,E1 -6208.373,E2 -6208.373} C_VEL
LIN {X 0,Y 494.898,Z 787.311,A -85,B 0,C 180,E1 -6210.001,E2 -6210.001} C_VEL
LIN {X 0,Y 494.962,Z 786.487,A -85,B 0,C 180,E1 -6211.628,E2 -6211.628} C_VEL
LIN {X 0,Y 494.998,Z 785.492,A -85,B 0,C 180,E1 -6212.442,E2 -6212.442} C_VEL
LIN {X 0,Y 495.042,Z 784.097,A -85,B 0,C 180,E1 -6213.256,E2 -6213.256} C_VEL
LIN {X 0,Y 495.016,Z 781.162,A -85,B 0,C 180,E1 -6214.479,E2 -6214.479} C_VEL
LIN {X 0,Y 495.16,Z 777.194,A -85,B 0,C 180,E1 -6215.703,E2 -6215.703} C_VEL
LIN {X 0,Y 495.258,Z 771.081,A -85,B 0,C 180,E1 -6217.133,E2 -6217.133} C_VEL
LIN {X 0,Y 495.447,Z 764.404,A -85,B 0,C 180,E1 -6218.361,E2 -6218.361} C_VEL
LIN {X 0,Y 495.732,Z 756.12,A -85,B 0,C 180,E1 -6219.59,E2 -6219.59} C_VEL
LIN {X 0,Y 496.014,Z 747.629,A -85,B 0,C 180,E1 -6220.615,E2 -6220.615} C_VEL
LIN {X 0,Y 496.475,Z 737.141,A -85,B 0,C 180,E1 -6221.638,E2 -6221.638} C_VEL
LIN {X 0,Y 496.789,Z 725.619,A -85,B 0,C 180,E1 -6222.542,E2 -6222.542} C_VEL
LIN {X 0,Y 497.225,Z 713.465,A -85,B 0,C 180,E1 -6223.279,E2 -6223.279} C_VEL
LIN {X 0,Y 497.61,Z 701.123,A -85,B 0,C 180,E1 -6223.841,E2 -6223.841} C_VEL
LIN {X 0,Y 497.924,Z 688.445,A -85,B 0,C 180,E1 -6224.249,E2 -6224.249} C_VEL
LIN {X 0,Y 498.137,Z 675.203,A -85,B 0,C 180,E1 -6224.503,E2 -6224.503} C_VEL
LIN {X 0,Y 498.421,Z 587.971,A -85,B 0,C 180,E1 -6225.769,E2 -6225.769} C_VEL
LIN {X 0,Y 496.382,Z 575.331,A -85,B 0,C 180,E1 -6226.031,E2 -6226.031} C_VEL
LIN {X 0,Y 496.364,Z 573.529,A -85,B 0,C 180,E1 -6226.241,E2 -6226.241} C_VEL
LIN {X 0,Y 496.917,Z 555.829,A -85,B 0,C 180,E1 -6229.198,E2 -6229.198} C_VEL
LIN {X 0,Y 497.585,Z 536.779,A -85,B 0,C 180,E1 -6232.418,E2 -6232.418} C_VEL
LIN {X 0,Y 497.523,Z 531.689,A -85,B 0,C 180,E1 -6233.299,E2 -6233.299} C_VEL
LIN {X 0,Y 495.83,Z 522.813,A -85,B 0,C 180,E1 -6234.979,E2 -6234.979} C_VEL
LIN {X 0,Y 495.783,Z 522.723,A -85,B 0,C 180,E1 -6237.892,E2 -6237.892} C_VEL
LIN {X 0,Y 495.756,Z 522.731,A -85,B 0,C 180,E1 -6240.688,E2 -6240.688} C_VEL
LIN {X 0,Y 495.763,Z 522.73,A -85,B 0,C 180,E1 -6243.565,E2 -6243.565} C_VEL
LIN {X 0,Y 495.732,Z 522.733,A -85,B 0,C 180,E1 -6246.544,E2 -6246.544} C_VEL
LIN {X 0,Y 495.76,Z 522.73,A -85,B 0,C 180,E1 -6249.638,E2 -6249.638} C_VEL
LIN {X 0,Y 495.742,Z 522.732,A -85,B 0,C 180,E1 -6252.507,E2 -6252.507} C_VEL
LIN {X 0,Y 495.754,Z 522.729,A -85,B 0,C 180,E1 -6255.14,E2 -6255.14} C_VEL
LIN {X 0,Y 495.762,Z 522.733,A -85,B 0,C 180,E1 -6258.219,E2 -6258.219} C_VEL
LIN {X 0,Y 495.755,Z 522.73,A -85,B 0,C 180,E1 -6261.409,E2 -6261.409} C_VEL
LIN {X 0,Y 495.762,Z 522.729,A -85,B 0,C 180,E1 -6264.463,E2 -6264.463} C_VEL
LIN {X 0,Y 495.772,Z 522.73,A -85,B 0,C 180,E1 -6267.406,E2 -6267.406} C_VEL
LIN {X 0,Y 495.77,Z 522.732,A -85,B 0,C 180,E1 -6270.254,E2 -6270.254} C_VEL
LIN {X 0,Y 495.867,Z 522.881,A -85,B 0,C 180,E1 -6273.477,E2 -6273.477} C_VEL
LIN {X 0,Y 497.692,Z 533.007,A -85,B 0,C 180,E1 -6274.936,E2 -6274.936} C_VEL
LIN {X 0,Y 497.384,Z 554.153,A -85,B 0,C 180,E1 -6277.792,E2 -6277.792} C_VEL
LIN {X 0,Y 496.978,Z 576.06,A -85,B 0,C 180,E1 -6280.805,E2 -6280.805} C_VEL
LIN {X 0,Y 496.489,Z 601.303,A -85,B 0,C 180,E1 -6284.275,E2 -6284.275} C_VEL
LIN {X 0,Y 496.007,Z 624.567,A -85,B 0,C 180,E1 -6287.521,E2 -6287.521} C_VEL
LIN {X 0,Y 495.939,Z 631.387,A -85,B 0,C 180,E1 -6288.435,E2 -6288.435} C_VEL
LIN {X 0,Y 496.837,Z 641.634,A -85,B 0,C 180,E1 -6288.629,E2 -6288.629} C_VEL
LIN {X 0,Y 496.521,Z 702.832,A -85,B 0,C 180,E1 -6289.577,E2 -6289.577} C_VEL
LIN {X 0,Y 496.425,Z 712.561,A -85,B 0,C 180,E1 -6289.858,E2 -6289.858} C_VEL
LIN {X 0,Y 496.241,Z 722.26,A -85,B 0,C 180,E1 -6290.267,E2 -6290.267} C_VEL
LIN {X 0,Y 496.056,Z 732.011,A -85,B 0,C 180,E1 -6290.829,E2 -6290.829} C_VEL
LIN {X 0,Y 495.761,Z 741.261,A -85,B 0,C 180,E1 -6291.542,E2 -6291.542} C_VEL
LIN {X 0,Y 495.574,Z 748.674,A -85,B 0,C 180,E1 -6292.257,E2 -6292.257} C_VEL
LIN {X 0,Y 495.43,Z 756.627,A -85,B 0,C 180,E1 -6293.218,E2 -6293.218} C_VEL
LIN {X 0,Y 495.309,Z 762.32,A -85,B 0,C 180,E1 -6294.095,E2 -6294.095} C_VEL
LIN {X 0,Y 495.109,Z 767.581,A -85,B 0,C 180,E1 -6295.114,E2 -6295.114} C_VEL
LIN {X 0,Y 495.126,Z 770.922,A -85,B 0,C 180,E1 -6295.93,E2 -6295.93} C_VEL
LIN {X 0,Y 495.027,Z 774.683,A -85,B 0,C 180,E1 -6297.152,E2 -6297.152} C_VEL
LIN {X 0,Y 494.961,Z 777.018,A -85,B 0,C 180,E1 -6298.373,E2 -6298.373} C_VEL
LIN {X 0,Y 494.907,Z 777.888,A -85,B 0,C 180,E1 -6299.186,E2 -6299.186} C_VEL
LIN {X 0,Y 494.897,Z 778.193,A -85,B 0,C 180,E1 -6300,E2 -6300} C_VEL
LIN {X 0,Y 494.909,Z 777.934,A -85,B 0,C 180,E1 -6300.814,E2 -6300.814} C_VEL
LIN {X 0,Y 494.962,Z 777.12,A -85,B 0,C 180,E1 -6301.627,E2 -6301.627} C_VEL
LIN {X 0,Y 495,Z 775.748,A -85,B 0,C 180,E1 -6302.441,E2 -6302.441} C_VEL
LIN {X 0,Y 495.101,Z 772.657,A -85,B 0,C 180,E1 -6303.662,E2 -6303.662} C_VEL
LIN {X 0,Y 495.09,Z 767.995,A -85,B 0,C 180,E1 -6304.886,E2 -6304.886} C_VEL
LIN {X 0,Y 495.304,Z 762.838,A -85,B 0,C 180,E1 -6305.905,E2 -6305.905} C_VEL
LIN {X 0,Y 495.422,Z 756.265,A -85,B 0,C 180,E1 -6306.925,E2 -6306.925} C_VEL
LIN {X 0,Y 495.554,Z 749.58,A -85,B 0,C 180,E1 -6307.743,E2 -6307.743} C_VEL
LIN {X 0,Y 495.798,Z 741.198,A -85,B 0,C 180,E1 -6308.56,E2 -6308.56} C_VEL
LIN {X 0,Y 496.067,Z 731.944,A -85,B 0,C 180,E1 -6309.274,E2 -6309.274} C_VEL
LIN {X 0,Y 496.279,Z 722.22,A -85,B 0,C 180,E1 -6309.836,E2 -6309.836} C_VEL
LIN {X 0,Y 496.396,Z 712.531,A -85,B 0,C 180,E1 -6310.245,E2 -6310.245} C_VEL
LIN {X 0,Y 496.569,Z 701.775,A -85,B 0,C 180,E1 -6310.551,E2 -6310.551} C_VEL
LIN {X 0,Y 496.751,Z 638.661,A -85,B 0,C 180,E1 -6311.513,E2 -6311.513} C_VEL
LIN {X 0,Y 495.915,Z 631.212,A -85,B 0,C 180,E1 -6311.67,E2 -6311.67} C_VEL
LIN {X 0,Y 496.351,Z 609.182,A -85,B 0,C 180,E1 -6314.766,E2 -6314.766} C_VEL
LIN {X 0,Y 496.861,Z 586.99,A -85,B 0,C 180,E1 -6317.918,E2 -6317.918} C_VEL
LIN {X 0,Y 497.453,Z 564.967,A -85,B 0,C 180,E1 -6321.057,E2 -6321.057} C_VEL
LIN {X 0,Y 497.995,Z 544.701,A -85,B 0,C 180,E1 -6323.943,E2 -6323.943} C_VEL
LIN {X 0,Y 498.092,Z 534.303,A -85,B 0,C 180,E1 -6325.44,E2 -6325.44} C_VEL
LIN {X 0,Y 495.826,Z 522.83,A -85,B 0,C 180,E1 -6327.23,E2 -6327.23} C_VEL
LIN {X 0,Y 495.769,Z 522.733,A -85,B 0,C 180,E1 -6330.147,E2 -6330.147} C_VEL
LIN {X 0,Y 495.798,Z 522.723,A -85,B 0,C 180,E1 -6333.244,E2 -6333.244} C_VEL
LIN {X 0,Y 495.734,Z 522.734,A -85,B 0,C 180,E1 -6336.09,E2 -6336.09} C_VEL
LIN {X 0,Y 495.769,Z 522.729,A -85,B 0,C 180,E1 -6338.768,E2 -6338.768} C_VEL
LIN {X 0,Y 495.761,Z 522.717,A -85,B 0,C 180,E1 -6341.781,E2 -6341.781} C_VEL
LIN {X 0,Y 495.754,Z 522.727,A -85,B 0,C 180,E1 -6345.139,E2 -6345.139} C_VEL
LIN {X 0,Y 495.727,Z 522.732,A -85,B 0,C 180,E1 -6346.716,E2 -6346.716} C_VEL
LIN {X 0,Y 495.069,Z 522.814,A -85,B 0,C 180,E1 -6347.394,E2 -6347.394} C_VEL
LIN {X 0,Y 492.226,Z 523.17,A -85,B 0,C 180,E1 -6348.494,E2 -6348.494} C_VEL
LIN {X 0,Y 489.818,Z 523.462,A -85,B 0,C 180,E1 -6349.381,E2 -6349.381} C_VEL
LIN {X 0,Y 488.783,Z 523.591,A -85,B 0,C 180,E1 -6350.066,E2 -6350.066} C_VEL
LIN {X 0,Y 488.698,Z 523.598,A -85,B 0,C 180,E1 -6350.298,E2 -6350.298} C_VEL
LIN {X 0,Y 488.687,Z 523.608,A -85,B 0,C 180,E1 -6353.645,E2 -6353.645} C_VEL
LIN {X 0,Y 488.739,Z 523.604,A -85,B 0,C 180,E1 -6356.516,E2 -6356.516} C_VEL
LIN {X 0,Y 488.729,Z 523.604,A -85,B 0,C 180,E1 -6359.78,E2 -6359.78} C_VEL
LIN {X 0,Y 488.797,Z 523.598,A -85,B 0,C 180,E1 -6363.056,E2 -6363.056} C_VEL
LIN {X 0,Y 488.682,Z 523.607,A -85,B 0,C 180,E1 -6366.253,E2 -6366.253} C_VEL
LIN {X 0,Y 488.77,Z 523.791,A -85,B 0,C 180,E1 -6368.6,E2 -6368.6} C_VEL
LIN {X 0,Y 489.922,Z 530.451,A -85,B 0,C 180,E1 -6370.08,E2 -6370.08} C_VEL
LIN {X 0,Y 489.464,Z 545.093,A -85,B 0,C 180,E1 -6373.096,E2 -6373.096} C_VEL
LIN {X 0,Y 489.361,Z 548.713,A -85,B 0,C 180,E1 -6373.771,E2 -6373.771} C_VEL
LIN {X 0,Y 491.786,Z 562.259,A -85,B 0,C 180,E1 -6374.083,E2 -6374.083} C_VEL
LIN {X 0,Y 491.211,Z 655.584,A -85,B 0,C 180,E1 -6375.473,E2 -6375.473} C_VEL
LIN {X 0,Y 490.919,Z 668.736,A -85,B 0,C 180,E1 -6375.834,E2 -6375.834} C_VEL
LIN {X 0,Y 490.606,Z 680.813,A -85,B 0,C 180,E1 -6376.327,E2 -6376.327} C_VEL
LIN {X 0,Y 490.275,Z 691.757,A -85,B 0,C 180,E1 -6376.924,E2 -6376.924} C_VEL
LIN {X 0,Y 489.93,Z 702.578,A -85,B 0,C 180,E1 -6377.679,E2 -6377.679} C_VEL
LIN {X 0,Y 489.464,Z 713.274,A -85,B 0,C 180,E1 -6378.613,E2 -6378.613} C_VEL
LIN {X 0,Y 489.087,Z 722.892,A -85,B 0,C 180,E1 -6379.652,E2 -6379.652} C_VEL
LIN {X 0,Y 488.737,Z 730.771,A -85,B 0,C 180,E1 -6380.689,E2 -6380.689} C_VEL
LIN {X 0,Y 488.455,Z 738.473,A -85,B 0,C 180,E1 -6381.935,E2 -6381.935} C_VEL
LIN {X 0,Y 488.183,Z 745.539,A -85,B 0,C 180,E1 -6383.386,E2 -6383.386} C_VEL
LIN {X 0,Y 488.073,Z 750.246,A -85,B 0,C 180,E1 -6384.629,E2 -6384.629} C_VEL
LIN {X 0,Y 488.068,Z 753.845,A -85,B 0,C 180,E1 -6385.871,E2 -6385.871} C_VEL
LIN {X 0,Y 487.979,Z 755.709,A -85,B 0,C 180,E1 -6386.697,E2 -6386.697} C_VEL
LIN {X 0,Y 487.933,Z 757.116,A -85,B 0,C 180,E1 -6387.523,E2 -6387.523} C_VEL
LIN {X 0,Y 487.834,Z 758.735,A -85,B 0,C 180,E1 -6389.174,E2 -6389.174} C_VEL
